Yaskawa INFORM job: DEMO_ROOF_UPPER_0625_3PAINT_23.JBI

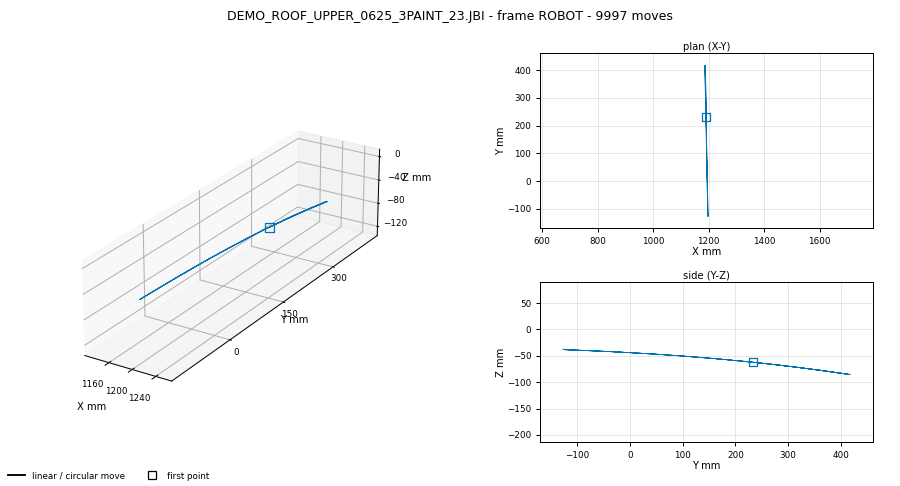
[picture p0: tool path of DEMO_ROOF_UPPER_0625_3PAINT_23.JBI in frame ROBOT, 9997 of 9997 moves have a stored position in this frame; points joined in program order, loops and branches not executed]
/JOB
//NAME DEMO_ROOF_UPPER_0625_3PAINT23
//POS
///NPOS 9997,0,0,0,0,0
///TOOL 0
///USER 0
///POSTYPE ROBOT
///RECTAN
///RCONF 1,0,0,0,0,0,0,0,0,0,0,0,0,0,0,0,0,0,0,0,0,0,0,0
C00000=1191.558,232.697,-61.990,-177.381,6.861,148.504
C00001=1191.554,232.946,-62.016,-177.379,6.863,148.503
C00002=1191.549,233.194,-62.041,-177.376,6.866,148.503
C00003=1191.545,233.443,-62.067,-177.373,6.868,148.503
C00004=1191.540,233.692,-62.093,-177.371,6.870,148.503
C00005=1191.536,233.941,-62.119,-177.368,6.873,148.503
C00006=1191.531,234.189,-62.145,-177.365,6.874,148.502
C00007=1191.527,234.437,-62.171,-177.363,6.877,148.502
C00008=1191.523,234.686,-62.197,-177.360,6.879,148.502
C00009=1191.519,234.935,-62.223,-177.358,6.881,148.502
C00010=1191.513,235.183,-62.249,-177.355,6.883,148.501
C00011=1191.509,235.432,-62.274,-177.352,6.886,148.501
C00012=1191.505,235.681,-62.300,-177.350,6.888,148.501
C00013=1191.500,235.929,-62.326,-177.348,6.890,148.501
C00014=1191.495,236.177,-62.353,-177.344,6.893,148.501
C00015=1191.490,236.449,-62.381,-177.342,6.895,148.500
C00016=1191.486,236.721,-62.409,-177.339,6.898,148.500
C00017=1191.481,236.992,-62.437,-177.336,6.900,148.500
C00018=1191.476,237.264,-62.465,-177.333,6.902,148.500
C00019=1191.471,237.512,-62.492,-177.330,6.905,148.500
C00020=1191.467,237.761,-62.518,-177.328,6.907,148.499
C00021=1191.463,238.010,-62.544,-177.326,6.909,148.499
C00022=1191.458,238.259,-62.570,-177.322,6.912,148.499
C00023=1191.453,238.506,-62.596,-177.320,6.914,148.499
C00024=1191.449,238.755,-62.622,-177.318,6.916,148.498
C00025=1191.444,239.004,-62.648,-177.315,6.919,148.498
C00026=1191.440,239.252,-62.675,-177.312,6.921,148.498
C00027=1191.436,239.501,-62.700,-177.310,6.923,148.498
C00028=1191.431,239.750,-62.727,-177.307,6.925,148.498
C00029=1191.427,239.998,-62.753,-177.305,6.928,148.498
C00030=1191.422,240.247,-62.779,-177.302,6.930,148.497
C00031=1191.418,240.495,-62.806,-177.299,6.932,148.497
C00032=1191.414,240.744,-62.831,-177.297,6.934,148.497
C00033=1191.409,240.993,-62.857,-177.294,6.937,148.497
C00034=1191.405,241.241,-62.884,-177.291,6.939,148.496
C00035=1191.400,241.490,-62.910,-177.289,6.941,148.496
C00036=1191.396,241.738,-62.937,-177.286,6.944,148.496
C00037=1191.392,241.987,-62.963,-177.284,6.946,148.496
C00038=1191.386,242.235,-62.989,-177.281,6.948,148.496
C00039=1191.382,242.484,-63.015,-177.279,6.951,148.496
C00040=1191.378,242.732,-63.042,-177.276,6.953,148.495
C00041=1191.373,242.981,-63.068,-177.273,6.956,148.495
C00042=1191.369,243.229,-63.094,-177.270,6.957,148.495
C00043=1191.364,243.478,-63.121,-177.268,6.960,148.495
C00044=1191.360,243.727,-63.147,-177.265,6.962,148.495
C00045=1191.355,243.976,-63.174,-177.263,6.964,148.494
C00046=1191.351,244.224,-63.200,-177.260,6.967,148.494
C00047=1191.347,244.473,-63.226,-177.258,6.969,148.494
C00048=1191.343,244.721,-63.253,-177.255,6.971,148.494
C00049=1191.338,244.970,-63.280,-177.252,6.974,148.494
C00050=1191.334,245.219,-63.306,-177.250,6.976,148.494
C00051=1191.329,245.467,-63.333,-177.247,6.979,148.493
C00052=1191.325,245.715,-63.359,-177.245,6.981,148.493
C00053=1191.320,245.964,-63.386,-177.242,6.983,148.493
C00054=1191.316,246.213,-63.412,-177.239,6.986,148.493
C00055=1191.312,246.461,-63.439,-177.237,6.988,148.493
C00056=1191.307,246.710,-63.465,-177.234,6.991,148.492
C00057=1191.303,246.958,-63.492,-177.231,6.992,148.492
C00058=1191.298,247.207,-63.519,-177.229,6.995,148.492
C00059=1191.294,247.456,-63.545,-177.226,6.998,148.492
C00060=1191.289,247.704,-63.572,-177.224,6.999,148.492
C00061=1191.285,247.953,-63.599,-177.221,7.002,148.492
C00062=1191.281,248.201,-63.625,-177.218,7.004,148.491
C00063=1191.276,248.450,-63.652,-177.216,7.006,148.491
C00064=1191.271,248.698,-63.679,-177.213,7.009,148.491
C00065=1191.267,248.947,-63.705,-177.211,7.011,148.491
C00066=1191.262,249.195,-63.732,-177.208,7.014,148.491
C00067=1191.258,249.443,-63.759,-177.206,7.016,148.490
C00068=1191.254,249.692,-63.786,-177.203,7.019,148.490
C00069=1191.249,249.941,-63.812,-177.200,7.021,148.490
C00070=1191.245,250.189,-63.839,-177.198,7.023,148.490
C00071=1191.240,250.438,-63.866,-177.195,7.026,148.490
C00072=1191.236,250.686,-63.893,-177.193,7.028,148.490
C00073=1191.231,250.935,-63.920,-177.190,7.031,148.490
C00074=1191.227,251.183,-63.946,-177.187,7.033,148.489
C00075=1191.222,251.431,-63.973,-177.185,7.036,148.489
C00076=1191.218,251.680,-64.000,-177.182,7.038,148.489
C00077=1191.214,251.928,-64.027,-177.179,7.041,148.489
C00078=1191.210,252.177,-64.054,-177.177,7.043,148.489
C00079=1191.205,252.426,-64.081,-177.174,7.045,148.488
C00080=1191.200,252.674,-64.108,-177.172,7.048,148.488
C00081=1191.196,252.923,-64.135,-177.170,7.050,148.488
C00082=1191.192,253.171,-64.162,-177.166,7.052,148.488
C00083=1191.187,253.419,-64.189,-177.164,7.055,148.488
C00084=1191.183,253.668,-64.216,-177.162,7.058,148.488
C00085=1191.178,253.916,-64.243,-177.159,7.059,148.488
C00086=1191.174,254.164,-64.270,-177.156,7.062,148.487
C00087=1191.170,254.414,-64.297,-177.154,7.064,148.487
C00088=1191.165,254.662,-64.324,-177.151,7.067,148.487
C00089=1191.161,254.911,-64.351,-177.149,7.069,148.487
C00090=1191.156,255.159,-64.378,-177.146,7.071,148.487
C00091=1191.151,255.408,-64.405,-177.143,7.074,148.487
C00092=1191.147,255.656,-64.432,-177.141,7.076,148.487
C00093=1191.143,255.905,-64.459,-177.138,7.079,148.486
C00094=1191.139,256.153,-64.487,-177.136,7.081,148.486
C00095=1191.134,256.401,-64.514,-177.133,7.084,148.486
C00096=1191.130,256.650,-64.541,-177.130,7.086,148.486
C00097=1191.125,256.898,-64.568,-177.128,7.089,148.486
C00098=1191.120,257.147,-64.595,-177.126,7.091,148.486
C00099=1191.117,257.395,-64.623,-177.122,7.094,148.485
C00100=1191.112,257.644,-64.650,-177.120,7.096,148.485
C00101=1191.107,257.892,-64.677,-177.117,7.099,148.485
C00102=1191.103,258.141,-64.704,-177.115,7.101,148.485
C00103=1191.099,258.388,-64.732,-177.112,7.104,148.485
C00104=1191.095,258.638,-64.759,-177.110,7.106,148.485
C00105=1191.090,258.886,-64.786,-177.107,7.109,148.485
C00106=1191.086,259.135,-64.813,-177.105,7.111,148.485
C00107=1191.081,259.383,-64.841,-177.102,7.114,148.484
C00108=1191.077,259.632,-64.868,-177.099,7.116,148.484
C00109=1191.073,259.880,-64.895,-177.097,7.119,148.484
C00110=1191.068,260.128,-64.923,-177.094,7.121,148.484
C00111=1191.064,260.377,-64.950,-177.091,7.123,148.484
C00112=1191.060,260.626,-64.978,-177.089,7.126,148.484
C00113=1191.055,260.874,-65.006,-177.086,7.129,148.484
C00114=1191.051,261.122,-65.033,-177.084,7.130,148.483
C00115=1191.046,261.370,-65.060,-177.081,7.133,148.483
C00116=1191.042,261.619,-65.088,-177.079,7.136,148.483
C00117=1191.037,261.867,-65.116,-177.076,7.139,148.483
C00118=1191.032,262.116,-65.143,-177.073,7.140,148.483
C00119=1191.028,262.389,-65.173,-177.071,7.143,148.483
C00120=1191.023,262.662,-65.204,-177.068,7.146,148.483
C00121=1191.019,262.935,-65.234,-177.065,7.149,148.482
C00122=1191.013,263.208,-65.265,-177.062,7.152,148.482
C00123=1191.009,263.456,-65.292,-177.059,7.154,148.482
C00124=1191.005,263.705,-65.320,-177.057,7.157,148.482
C00125=1191.000,263.953,-65.347,-177.055,7.159,148.482
C00126=1190.996,264.201,-65.375,-177.052,7.162,148.482
C00127=1190.992,264.450,-65.402,-177.049,7.164,148.482
C00128=1190.987,264.698,-65.430,-177.046,7.167,148.482
C00129=1190.983,264.946,-65.458,-177.044,7.169,148.481
C00130=1190.978,265.195,-65.486,-177.042,7.172,148.481
C00131=1190.974,265.443,-65.513,-177.038,7.175,148.481
C00132=1190.969,265.692,-65.540,-177.036,7.177,148.481
C00133=1190.966,265.940,-65.569,-177.034,7.180,148.481
C00134=1190.961,266.188,-65.596,-177.031,7.182,148.481
C00135=1190.956,266.437,-65.624,-177.028,7.185,148.481
C00136=1190.952,266.686,-65.652,-177.026,7.187,148.481
C00137=1190.948,266.934,-65.680,-177.023,7.190,148.481
C00138=1190.944,267.183,-65.707,-177.021,7.192,148.480
C00139=1190.939,267.431,-65.736,-177.018,7.195,148.480
C00140=1190.934,267.679,-65.764,-177.015,7.198,148.480
C00141=1190.930,267.927,-65.792,-177.013,7.200,148.480
C00142=1190.926,268.176,-65.819,-177.010,7.203,148.480
C00143=1190.921,268.425,-65.848,-177.008,7.205,148.480
C00144=1190.917,268.673,-65.875,-177.005,7.208,148.480
C00145=1190.913,268.920,-65.903,-177.003,7.210,148.480
C00146=1190.909,269.170,-65.930,-177.000,7.213,148.480
C00147=1190.903,269.418,-65.959,-176.998,7.215,148.479
C00148=1190.900,269.666,-65.987,-176.995,7.218,148.479
C00149=1190.895,269.914,-66.015,-176.992,7.221,148.479
C00150=1190.891,270.163,-66.044,-176.990,7.223,148.479
C00151=1190.887,270.411,-66.071,-176.987,7.226,148.479
C00152=1190.882,270.660,-66.099,-176.985,7.228,148.479
C00153=1190.877,270.908,-66.127,-176.982,7.231,148.479
C00154=1190.874,271.157,-66.155,-176.980,7.233,148.479
C00155=1190.869,271.405,-66.183,-176.977,7.236,148.479
C00156=1190.864,271.653,-66.211,-176.974,7.239,148.479
C00157=1190.860,271.902,-66.240,-176.972,7.241,148.478
C00158=1190.855,272.150,-66.268,-176.969,7.244,148.478
C00159=1190.852,272.398,-66.296,-176.967,7.246,148.478
C00160=1190.847,272.646,-66.324,-176.964,7.249,148.478
C00161=1190.843,272.895,-66.353,-176.961,7.252,148.478
C00162=1190.838,273.143,-66.380,-176.959,7.254,148.478
C00163=1190.834,273.392,-66.409,-176.956,7.257,148.478
C00164=1190.830,273.640,-66.437,-176.954,7.259,148.478
C00165=1190.825,273.889,-66.466,-176.951,7.262,148.478
C00166=1190.821,274.137,-66.494,-176.948,7.265,148.478
C00167=1190.817,274.385,-66.522,-176.946,7.267,148.477
C00168=1190.813,274.634,-66.550,-176.943,7.270,148.477
C00169=1190.808,274.882,-66.578,-176.941,7.272,148.477
C00170=1190.804,275.131,-66.607,-176.938,7.275,148.477
C00171=1190.799,275.379,-66.635,-176.936,7.278,148.477
C00172=1190.795,275.627,-66.664,-176.933,7.280,148.477
C00173=1190.791,275.875,-66.692,-176.931,7.283,148.477
C00174=1190.786,276.124,-66.721,-176.928,7.285,148.477
C00175=1190.783,276.372,-66.749,-176.925,7.288,148.477
C00176=1190.777,276.621,-66.777,-176.923,7.291,148.477
C00177=1190.773,276.869,-66.806,-176.920,7.293,148.477
C00178=1190.769,277.117,-66.834,-176.918,7.296,148.476
C00179=1190.764,277.366,-66.863,-176.915,7.299,148.476
C00180=1190.760,277.613,-66.891,-176.913,7.301,148.476
C00181=1190.756,277.862,-66.920,-176.910,7.304,148.476
C00182=1190.752,278.111,-66.948,-176.908,7.306,148.476
C00183=1190.747,278.358,-66.977,-176.905,7.309,148.476
C00184=1190.743,278.607,-67.005,-176.902,7.312,148.476
C00185=1190.739,278.856,-67.034,-176.900,7.314,148.476
C00186=1190.734,279.103,-67.063,-176.897,7.317,148.476
C00187=1190.730,279.352,-67.091,-176.895,7.320,148.476
C00188=1190.725,279.600,-67.119,-176.892,7.322,148.476
C00189=1190.721,279.849,-67.148,-176.889,7.325,148.475
C00190=1190.717,280.097,-67.177,-176.887,7.327,148.475
C00191=1190.712,280.345,-67.205,-176.884,7.330,148.475
C00192=1190.708,280.594,-67.235,-176.882,7.333,148.475
C00193=1190.704,280.842,-67.263,-176.879,7.335,148.475
C00194=1190.699,281.090,-67.291,-176.877,7.338,148.475
C00195=1190.695,281.339,-67.321,-176.874,7.341,148.475
C00196=1190.691,281.587,-67.349,-176.872,7.344,148.475
C00197=1190.686,281.835,-67.378,-176.869,7.347,148.475
C00198=1190.682,282.084,-67.407,-176.866,7.349,148.475
C00199=1190.678,282.332,-67.435,-176.864,7.351,148.475
C00200=1190.673,282.580,-67.464,-176.861,7.354,148.475
C00201=1190.669,282.829,-67.493,-176.858,7.357,148.475
C00202=1190.665,283.077,-67.522,-176.856,7.360,148.475
C00203=1190.661,283.325,-67.550,-176.854,7.363,148.475
C00204=1190.656,283.573,-67.579,-176.851,7.366,148.475
C00205=1190.652,283.822,-67.608,-176.849,7.368,148.474
C00206=1190.648,284.070,-67.637,-176.846,7.371,148.474
C00207=1190.643,284.318,-67.667,-176.843,7.374,148.474
C00208=1190.639,284.566,-67.695,-176.841,7.376,148.474
C00209=1190.635,284.815,-67.724,-176.838,7.379,148.474
C00210=1190.630,285.064,-67.753,-176.835,7.382,148.474
C00211=1190.626,285.311,-67.782,-176.833,7.384,148.474
C00212=1190.621,285.559,-67.811,-176.830,7.387,148.474
C00213=1190.617,285.808,-67.840,-176.828,7.390,148.474
C00214=1190.613,286.056,-67.869,-176.825,7.392,148.474
C00215=1190.608,286.304,-67.897,-176.823,7.395,148.474
C00216=1190.604,286.553,-67.927,-176.820,7.398,148.474
C00217=1190.600,286.801,-67.956,-176.818,7.400,148.474
C00218=1190.596,287.049,-67.986,-176.815,7.403,148.474
C00219=1190.591,287.298,-68.014,-176.812,7.406,148.474
C00220=1190.587,287.546,-68.044,-176.810,7.408,148.474
C00221=1190.582,287.794,-68.073,-176.808,7.411,148.474
C00222=1190.579,288.042,-68.101,-176.805,7.414,148.474
C00223=1190.573,288.317,-68.134,-176.802,7.417,148.474
C00224=1190.569,288.592,-68.166,-176.799,7.420,148.473
C00225=1190.564,288.866,-68.199,-176.796,7.423,148.473
C00226=1190.559,289.140,-68.231,-176.794,7.426,148.473
C00227=1190.555,289.388,-68.260,-176.791,7.429,148.473
C00228=1190.551,289.637,-68.290,-176.789,7.431,148.473
C00229=1190.546,289.885,-68.318,-176.786,7.434,148.473
C00230=1190.542,290.134,-68.348,-176.783,7.437,148.473
C00231=1190.538,290.382,-68.377,-176.781,7.439,148.473
C00232=1190.533,290.630,-68.406,-176.778,7.442,148.473
C00233=1190.529,290.878,-68.436,-176.776,7.445,148.473
C00234=1190.525,291.126,-68.465,-176.773,7.448,148.473
C00235=1190.521,291.374,-68.495,-176.771,7.451,148.473
C00236=1190.516,291.623,-68.524,-176.768,7.454,148.473
C00237=1190.512,291.871,-68.554,-176.765,7.457,148.473
C00238=1190.508,292.119,-68.583,-176.763,7.459,148.473
C00239=1190.504,292.367,-68.612,-176.761,7.462,148.473
C00240=1190.500,292.616,-68.642,-176.758,7.465,148.473
C00241=1190.495,292.863,-68.671,-176.755,7.468,148.473
C00242=1190.491,293.111,-68.700,-176.753,7.470,148.473
C00243=1190.487,293.360,-68.730,-176.750,7.473,148.473
C00244=1190.482,293.608,-68.759,-176.748,7.476,148.473
C00245=1190.477,293.857,-68.789,-176.745,7.478,148.472
C00246=1190.473,294.105,-68.819,-176.743,7.481,148.472
C00247=1190.469,294.353,-68.848,-176.740,7.484,148.472
C00248=1190.465,294.601,-68.878,-176.738,7.487,148.473
C00249=1190.461,294.850,-68.907,-176.736,7.490,148.473
C00250=1190.457,295.098,-68.937,-176.733,7.493,148.472
C00251=1190.452,295.346,-68.966,-176.730,7.496,148.472
C00252=1190.448,295.594,-68.996,-176.728,7.498,148.472
C00253=1190.443,295.843,-69.026,-176.725,7.501,148.472
C00254=1190.439,296.091,-69.056,-176.723,7.504,148.472
C00255=1190.435,296.339,-69.085,-176.720,7.507,148.472
C00256=1190.431,296.587,-69.115,-176.718,7.509,148.472
C00257=1190.427,296.836,-69.144,-176.715,7.512,148.472
C00258=1190.422,297.084,-69.174,-176.712,7.515,148.472
C00259=1190.418,297.332,-69.204,-176.710,7.518,148.472
C00260=1190.414,297.580,-69.234,-176.707,7.520,148.472
C00261=1190.410,297.828,-69.263,-176.705,7.523,148.472
C00262=1190.406,298.077,-69.293,-176.702,7.526,148.472
C00263=1190.401,298.324,-69.324,-176.699,7.529,148.472
C00264=1190.397,298.573,-69.353,-176.697,7.531,148.472
C00265=1190.393,298.821,-69.382,-176.695,7.535,148.472
C00266=1190.388,299.069,-69.413,-176.692,7.538,148.472
C00267=1190.384,299.317,-69.443,-176.690,7.541,148.472
C00268=1190.380,299.566,-69.472,-176.687,7.543,148.472
C00269=1190.376,299.813,-69.502,-176.685,7.546,148.472
C00270=1190.371,300.062,-69.532,-176.682,7.549,148.472
C00271=1190.367,300.310,-69.562,-176.679,7.552,148.472
C00272=1190.363,300.558,-69.592,-176.677,7.554,148.472
C00273=1190.358,300.806,-69.622,-176.674,7.557,148.472
C00274=1190.354,301.055,-69.651,-176.672,7.560,148.472
C00275=1190.350,301.302,-69.682,-176.669,7.563,148.472
C00276=1190.345,301.551,-69.712,-176.667,7.566,148.472
C00277=1190.341,301.798,-69.742,-176.665,7.569,148.472
C00278=1190.337,302.047,-69.771,-176.662,7.572,148.472
C00279=1190.332,302.295,-69.802,-176.659,7.575,148.472
C00280=1190.328,302.543,-69.832,-176.657,7.577,148.472
C00281=1190.324,302.792,-69.863,-176.654,7.580,148.472
C00282=1190.320,303.040,-69.892,-176.652,7.583,148.472
C00283=1190.315,303.288,-69.923,-176.649,7.586,148.472
C00284=1190.311,303.536,-69.952,-176.647,7.588,148.472
C00285=1190.307,303.784,-69.982,-176.644,7.591,148.472
C00286=1190.302,304.032,-70.013,-176.642,7.594,148.472
C00287=1190.298,304.280,-70.043,-176.639,7.597,148.472
C00288=1190.294,304.528,-70.073,-176.637,7.600,148.472
C00289=1190.289,304.776,-70.103,-176.634,7.603,148.472
C00290=1190.285,305.025,-70.134,-176.632,7.606,148.472
C00291=1190.281,305.273,-70.163,-176.629,7.609,148.472
C00292=1190.277,305.521,-70.194,-176.627,7.612,148.472
C00293=1190.273,305.769,-70.224,-176.624,7.614,148.472
C00294=1190.268,306.017,-70.254,-176.622,7.617,148.472
C00295=1190.264,306.265,-70.285,-176.619,7.620,148.472
C00296=1190.260,306.514,-70.316,-176.617,7.623,148.472
C00297=1190.256,306.762,-70.345,-176.615,7.626,148.472
C00298=1190.251,307.010,-70.376,-176.612,7.629,148.472
C00299=1190.247,307.257,-70.406,-176.609,7.632,148.472
C00300=1190.243,307.505,-70.437,-176.606,7.635,148.472
C00301=1190.238,307.754,-70.467,-176.604,7.638,148.472
C00302=1190.235,308.002,-70.498,-176.602,7.640,148.472
C00303=1190.230,308.250,-70.528,-176.599,7.643,148.472
C00304=1190.226,308.498,-70.558,-176.597,7.646,148.472
C00305=1190.221,308.746,-70.589,-176.594,7.649,148.472
C00306=1190.217,308.994,-70.619,-176.592,7.652,148.472
C00307=1190.213,309.243,-70.650,-176.590,7.655,148.472
C00308=1190.209,309.491,-70.681,-176.587,7.658,148.472
C00309=1190.205,309.738,-70.711,-176.584,7.661,148.472
C00310=1190.200,309.986,-70.741,-176.582,7.664,148.472
C00311=1190.196,310.235,-70.773,-176.579,7.667,148.472
C00312=1190.192,310.483,-70.803,-176.577,7.669,148.472
C00313=1190.187,310.731,-70.833,-176.574,7.672,148.472
C00314=1190.183,310.979,-70.864,-176.572,7.675,148.473
C00315=1190.179,311.228,-70.894,-176.569,7.678,148.473
C00316=1190.175,311.475,-70.925,-176.567,7.681,148.473
C00317=1190.170,311.723,-70.956,-176.565,7.684,148.472
C00318=1190.166,311.971,-70.986,-176.562,7.687,148.473
C00319=1190.162,312.220,-71.017,-176.560,7.690,148.473
C00320=1190.158,312.468,-71.048,-176.557,7.693,148.473
C00321=1190.153,312.716,-71.078,-176.554,7.696,148.473
C00322=1190.150,312.964,-71.109,-176.553,7.698,148.473
C00323=1190.145,313.212,-71.140,-176.550,7.701,148.473
C00324=1190.141,313.460,-71.171,-176.547,7.704,148.473
C00325=1190.137,313.709,-71.202,-176.544,7.707,148.473
C00326=1190.133,313.956,-71.232,-176.542,7.711,148.473
C00327=1190.127,314.232,-71.267,-176.539,7.714,148.473
C00328=1190.123,314.509,-71.301,-176.537,7.717,148.473
C00329=1190.119,314.786,-71.335,-176.534,7.720,148.473
C00330=1190.114,315.062,-71.370,-176.531,7.724,148.473
C00331=1190.110,315.310,-71.401,-176.529,7.726,148.473
C00332=1190.105,315.558,-71.431,-176.526,7.729,148.473
C00333=1190.101,315.806,-71.463,-176.524,7.733,148.473
C00334=1190.097,316.054,-71.494,-176.521,7.736,148.473
C00335=1190.093,316.302,-71.524,-176.519,7.739,148.473
C00336=1190.088,316.550,-71.555,-176.517,7.741,148.473
C00337=1190.084,316.799,-71.586,-176.514,7.744,148.473
C00338=1190.080,317.046,-71.618,-176.512,7.747,148.473
C00339=1190.075,317.294,-71.648,-176.509,7.750,148.473
C00340=1190.071,317.543,-71.680,-176.507,7.753,148.474
C00341=1190.067,317.791,-71.710,-176.504,7.756,148.474
C00342=1190.064,318.038,-71.742,-176.502,7.759,148.474
C00343=1190.059,318.286,-71.772,-176.500,7.762,148.474
C00344=1190.055,318.534,-71.803,-176.497,7.765,148.474
C00345=1190.051,318.782,-71.835,-176.495,7.768,148.474
C00346=1190.046,319.030,-71.866,-176.492,7.771,148.474
C00347=1190.042,319.279,-71.897,-176.490,7.773,148.474
C00348=1190.038,319.526,-71.928,-176.488,7.777,148.474
C00349=1190.034,319.775,-71.959,-176.485,7.780,148.474
C00350=1190.030,320.022,-71.991,-176.483,7.783,148.474
C00351=1190.026,320.271,-72.022,-176.480,7.786,148.474
C00352=1190.021,320.519,-72.053,-176.477,7.789,148.474
C00353=1190.017,320.766,-72.084,-176.476,7.792,148.474
C00354=1190.013,321.015,-72.115,-176.473,7.795,148.474
C00355=1190.008,321.262,-72.147,-176.471,7.798,148.475
C00356=1190.004,321.511,-72.178,-176.468,7.801,148.475
C00357=1190.000,321.758,-72.209,-176.465,7.804,148.475
C00358=1189.996,322.007,-72.241,-176.463,7.807,148.475
C00359=1189.992,322.254,-72.272,-176.461,7.809,148.475
C00360=1189.988,322.503,-72.303,-176.459,7.813,148.475
C00361=1189.983,322.750,-72.335,-176.456,7.816,148.475
C00362=1189.979,322.999,-72.366,-176.453,7.819,148.475
C00363=1189.975,323.246,-72.397,-176.451,7.822,148.475
C00364=1189.971,323.495,-72.428,-176.448,7.825,148.475
C00365=1189.967,323.742,-72.460,-176.446,7.828,148.475
C00366=1189.963,323.990,-72.492,-176.444,7.831,148.475
C00367=1189.958,324.238,-72.523,-176.442,7.834,148.476
C00368=1189.954,324.486,-72.555,-176.439,7.837,148.476
C00369=1189.950,324.735,-72.586,-176.437,7.840,148.476
C00370=1189.946,324.982,-72.618,-176.434,7.843,148.476
C00371=1189.942,325.231,-72.649,-176.432,7.847,148.476
C00372=1189.937,325.478,-72.680,-176.430,7.849,148.476
C00373=1189.934,325.727,-72.712,-176.427,7.852,148.476
C00374=1189.929,325.974,-72.744,-176.425,7.855,148.476
C00375=1189.925,326.222,-72.776,-176.422,7.858,148.476
C00376=1189.920,326.470,-72.807,-176.420,7.861,148.476
C00377=1189.917,326.718,-72.839,-176.417,7.865,148.477
C00378=1189.913,326.966,-72.870,-176.415,7.867,148.477
C00379=1189.909,327.214,-72.902,-176.413,7.870,148.477
C00380=1189.904,327.463,-72.934,-176.410,7.873,148.477
C00381=1189.900,327.710,-72.965,-176.408,7.877,148.477
C00382=1189.896,327.958,-72.997,-176.405,7.880,148.477
C00383=1189.892,328.206,-73.029,-176.403,7.883,148.477
C00384=1189.888,328.453,-73.060,-176.400,7.886,148.477
C00385=1189.883,328.702,-73.092,-176.399,7.888,148.477
C00386=1189.879,328.950,-73.123,-176.396,7.892,148.478
C00387=1189.875,329.198,-73.155,-176.394,7.895,148.478
C00388=1189.871,329.446,-73.187,-176.392,7.898,148.478
C00389=1189.866,329.693,-73.219,-176.389,7.901,148.478
C00390=1189.863,329.941,-73.251,-176.387,7.904,148.478
C00391=1189.859,330.189,-73.283,-176.384,7.907,148.478
C00392=1189.854,330.437,-73.315,-176.382,7.910,148.478
C00393=1189.850,330.685,-73.347,-176.380,7.913,148.478
C00394=1189.846,330.932,-73.378,-176.377,7.916,148.478
C00395=1189.841,331.181,-73.411,-176.375,7.920,148.479
C00396=1189.837,331.429,-73.442,-176.372,7.923,148.479
C00397=1189.833,331.677,-73.473,-176.370,7.926,148.479
C00398=1189.829,331.925,-73.506,-176.368,7.929,148.479
C00399=1189.825,332.173,-73.538,-176.366,7.931,148.479
C00400=1189.821,332.421,-73.570,-176.363,7.935,148.479
C00401=1189.816,332.668,-73.602,-176.361,7.938,148.479
C00402=1189.813,332.916,-73.634,-176.358,7.941,148.479
C00403=1189.808,333.165,-73.667,-176.356,7.944,148.480
C00404=1189.804,333.412,-73.698,-176.354,7.948,148.480
C00405=1189.800,333.660,-73.730,-176.351,7.951,148.480
C00406=1189.796,333.908,-73.762,-176.349,7.954,148.480
C00407=1189.792,334.156,-73.794,-176.347,7.957,148.480
C00408=1189.787,334.404,-73.826,-176.345,7.960,148.480
C00409=1189.783,334.652,-73.858,-176.342,7.963,148.480
C00410=1189.779,334.900,-73.891,-176.340,7.966,148.481
C00411=1189.775,335.147,-73.923,-176.337,7.969,148.481
C00412=1189.770,335.395,-73.955,-176.335,7.973,148.481
C00413=1189.767,335.644,-73.987,-176.333,7.976,148.481
C00414=1189.762,335.892,-74.019,-176.331,7.978,148.481
C00415=1189.758,336.139,-74.052,-176.329,7.981,148.481
C00416=1189.754,336.387,-74.084,-176.326,7.985,148.481
C00417=1189.750,336.635,-74.116,-176.324,7.988,148.482
C00418=1189.746,336.883,-74.148,-176.321,7.991,148.482
C00419=1189.742,337.130,-74.181,-176.319,7.994,148.482
C00420=1189.737,337.378,-74.213,-176.317,7.998,148.482
C00421=1189.734,337.626,-74.245,-176.315,8.001,148.482
C00422=1189.729,337.875,-74.277,-176.313,8.003,148.482
C00423=1189.726,338.122,-74.310,-176.310,8.007,148.482
C00424=1189.721,338.370,-74.342,-176.308,8.010,148.483
C00425=1189.717,338.617,-74.374,-176.306,8.013,148.483
C00426=1189.713,338.866,-74.407,-176.304,8.017,148.483
C00427=1189.708,339.114,-74.439,-176.301,8.020,148.483
C00428=1189.705,339.361,-74.472,-176.299,8.023,148.483
C00429=1189.701,339.610,-74.504,-176.296,8.026,148.484
C00430=1189.696,339.857,-74.536,-176.295,8.029,148.484
C00431=1189.691,340.136,-74.573,-176.292,8.033,148.484
C00432=1189.687,340.415,-74.610,-176.289,8.036,148.484
C00433=1189.682,340.693,-74.646,-176.287,8.039,148.484
C00434=1189.678,340.972,-74.683,-176.284,8.043,148.484
C00435=1189.673,341.220,-74.715,-176.282,8.047,148.485
C00436=1189.670,341.467,-74.748,-176.280,8.050,148.485
C00437=1189.665,341.716,-74.780,-176.278,8.053,148.485
C00438=1189.661,341.963,-74.813,-176.276,8.056,148.485
C00439=1189.657,342.212,-74.846,-176.273,8.059,148.486
C00440=1189.653,342.459,-74.878,-176.271,8.062,148.486
C00441=1189.648,342.707,-74.910,-176.268,8.065,148.486
C00442=1189.644,342.955,-74.944,-176.266,8.069,148.486
C00443=1189.641,343.203,-74.975,-176.264,8.072,148.486
C00444=1189.636,343.450,-75.009,-176.262,8.075,148.486
C00445=1189.632,343.698,-75.042,-176.260,8.079,148.487
C00446=1189.628,343.946,-75.074,-176.258,8.081,148.487
C00447=1189.624,344.194,-75.107,-176.256,8.085,148.487
C00448=1189.620,344.442,-75.140,-176.253,8.088,148.487
C00449=1189.615,344.689,-75.172,-176.251,8.091,148.487
C00450=1189.611,344.937,-75.205,-176.249,8.095,148.488
C00451=1189.607,345.185,-75.238,-176.247,8.098,148.488
C00452=1189.603,345.433,-75.270,-176.244,8.101,148.488
C00453=1189.599,345.680,-75.303,-176.242,8.105,148.488
C00454=1189.595,345.928,-75.336,-176.240,8.107,148.489
C00455=1189.591,346.177,-75.369,-176.238,8.110,148.489
C00456=1189.586,346.424,-75.402,-176.236,8.114,148.489
C00457=1189.583,346.672,-75.435,-176.234,8.117,148.489
C00458=1189.579,346.919,-75.468,-176.231,8.120,148.489
C00459=1189.574,347.168,-75.500,-176.229,8.124,148.490
C00460=1189.570,347.416,-75.533,-176.227,8.127,148.490
C00461=1189.566,347.663,-75.566,-176.225,8.130,148.490
C00462=1189.562,347.911,-75.600,-176.222,8.134,148.490
C00463=1189.558,348.159,-75.633,-176.221,8.136,148.490
C00464=1189.554,348.406,-75.666,-176.219,8.139,148.491
C00465=1189.550,348.654,-75.698,-176.216,8.143,148.491
C00466=1189.546,348.902,-75.731,-176.214,8.146,148.491
C00467=1189.542,349.150,-75.764,-176.212,8.150,148.492
C00468=1189.538,349.398,-75.797,-176.210,8.153,148.492
C00469=1189.533,349.645,-75.830,-176.208,8.156,148.492
C00470=1189.529,349.893,-75.864,-176.205,8.160,148.492
C00471=1189.525,350.141,-75.897,-176.203,8.163,148.492
C00472=1189.521,350.389,-75.930,-176.202,8.166,148.493
C00473=1189.517,350.636,-75.963,-176.199,8.169,148.493
C00474=1189.513,350.884,-75.996,-176.198,8.172,148.493
C00475=1189.509,351.132,-76.029,-176.195,8.176,148.493
C00476=1189.504,351.379,-76.063,-176.193,8.179,148.494
C00477=1189.500,351.627,-76.096,-176.191,8.182,148.494
C00478=1189.496,351.875,-76.129,-176.189,8.186,148.494
C00479=1189.492,352.123,-76.162,-176.187,8.189,148.495
C00480=1189.488,352.370,-76.195,-176.184,8.193,148.495
C00481=1189.484,352.618,-76.228,-176.183,8.195,148.495
C00482=1189.480,352.866,-76.261,-176.181,8.199,148.495
C00483=1189.476,353.114,-76.295,-176.179,8.202,148.496
C00484=1189.472,353.362,-76.328,-176.177,8.205,148.496
C00485=1189.468,353.610,-76.361,-176.174,8.209,148.496
C00486=1189.464,353.857,-76.394,-176.172,8.212,148.496
C00487=1189.460,354.105,-76.428,-176.170,8.216,148.497
C00488=1189.456,354.352,-76.461,-176.168,8.219,148.497
C00489=1189.452,354.600,-76.495,-176.166,8.222,148.497
C00490=1189.447,354.848,-76.528,-176.165,8.225,148.498
C00491=1189.443,355.096,-76.562,-176.162,8.229,148.498
C00492=1189.438,355.344,-76.595,-176.160,8.232,148.498
C00493=1189.435,355.591,-76.629,-176.158,8.235,148.498
C00494=1189.431,355.839,-76.662,-176.156,8.239,148.499
C00495=1189.427,356.087,-76.695,-176.154,8.242,148.499
C00496=1189.423,356.335,-76.728,-176.152,8.246,148.499
C00497=1189.419,356.582,-76.762,-176.150,8.249,148.500
C00498=1189.415,356.829,-76.795,-176.148,8.253,148.500
C00499=1189.410,357.077,-76.829,-176.146,8.255,148.500
C00500=1189.406,357.326,-76.863,-176.144,8.259,148.500
C00501=1189.403,357.573,-76.897,-176.142,8.262,148.501
C00502=1189.398,357.821,-76.930,-176.140,8.265,148.501
C00503=1189.394,358.068,-76.963,-176.138,8.269,148.501
C00504=1189.390,358.316,-76.997,-176.136,8.272,148.502
C00505=1189.386,358.564,-77.030,-176.134,8.276,148.502
C00506=1189.382,358.812,-77.064,-176.132,8.279,148.502
C00507=1189.378,359.059,-77.098,-176.130,8.283,148.503
C00508=1189.374,359.307,-77.131,-176.128,8.286,148.503
C00509=1189.370,359.554,-77.165,-176.127,8.289,148.503
C00510=1189.365,359.802,-77.199,-176.124,8.292,148.504
C00511=1189.362,360.050,-77.232,-176.122,8.296,148.504
C00512=1189.358,360.298,-77.266,-176.121,8.300,148.504
C00513=1189.353,360.546,-77.300,-176.118,8.303,148.505
C00514=1189.349,360.793,-77.334,-176.117,8.306,148.505
C00515=1189.346,361.041,-77.367,-176.115,8.309,148.505
C00516=1189.342,361.288,-77.401,-176.113,8.313,148.506
C00517=1189.337,361.536,-77.435,-176.111,8.316,148.506
C00518=1189.333,361.783,-77.469,-176.109,8.320,148.506
C00519=1189.330,362.032,-77.502,-176.107,8.323,148.507
C00520=1189.325,362.279,-77.537,-176.106,8.326,148.507
C00521=1189.321,362.527,-77.570,-176.104,8.330,148.507
C00522=1189.317,362.774,-77.604,-176.102,8.333,148.508
C00523=1189.313,363.023,-77.638,-176.100,8.337,148.508
C00524=1189.309,363.270,-77.672,-176.099,8.340,148.509
C00525=1189.305,363.517,-77.706,-176.097,8.343,148.509
C00526=1189.300,363.765,-77.739,-176.095,8.347,148.509
C00527=1189.297,364.013,-77.774,-176.093,8.350,148.510
C00528=1189.293,364.260,-77.807,-176.092,8.353,148.510
C00529=1189.288,364.508,-77.841,-176.090,8.357,148.511
C00530=1189.285,364.756,-77.875,-176.088,8.360,148.511
C00531=1189.281,365.004,-77.909,-176.086,8.364,148.511
C00532=1189.276,365.251,-77.943,-176.085,8.366,148.512
C00533=1189.273,365.499,-77.977,-176.083,8.370,148.512
C00534=1189.269,365.746,-78.012,-176.081,8.374,148.513
C00535=1189.264,366.027,-78.050,-176.079,8.377,148.513
C00536=1189.259,366.309,-78.088,-176.078,8.381,148.513
C00537=1189.255,366.590,-78.127,-176.076,8.384,148.514
C00538=1189.251,366.871,-78.166,-176.073,8.389,148.514
C00539=1189.247,367.119,-78.201,-176.072,8.392,148.515
C00540=1189.242,367.367,-78.234,-176.070,8.395,148.515
C00541=1189.238,367.614,-78.268,-176.069,8.399,148.516
C00542=1189.235,367.862,-78.302,-176.067,8.402,148.516
C00543=1189.230,368.109,-78.337,-176.066,8.405,148.516
C00544=1189.226,368.357,-78.370,-176.064,8.409,148.517
C00545=1189.222,368.605,-78.405,-176.063,8.412,148.517
C00546=1189.218,368.852,-78.439,-176.061,8.416,148.518
C00547=1189.214,369.100,-78.473,-176.060,8.419,148.518
C00548=1189.210,369.347,-78.507,-176.058,8.422,148.519
C00549=1189.206,369.595,-78.542,-176.056,8.426,148.519
C00550=1189.202,369.842,-78.576,-176.055,8.429,148.520
C00551=1189.198,370.091,-78.610,-176.053,8.432,148.520
C00552=1189.194,370.338,-78.644,-176.052,8.435,148.520
C00553=1189.190,370.586,-78.679,-176.051,8.439,148.521
C00554=1189.186,370.833,-78.712,-176.049,8.443,148.521
C00555=1189.181,371.080,-78.747,-176.048,8.445,148.522
C00556=1189.178,371.329,-78.782,-176.046,8.449,148.522
C00557=1189.174,371.576,-78.816,-176.045,8.452,148.523
C00558=1189.170,371.824,-78.850,-176.043,8.456,148.523
C00559=1189.166,372.071,-78.884,-176.042,8.459,148.524
C00560=1189.161,372.318,-78.919,-176.040,8.462,148.524
C00561=1189.158,372.566,-78.953,-176.039,8.465,148.525
C00562=1189.154,372.814,-78.988,-176.038,8.469,148.525
C00563=1189.150,373.062,-79.022,-176.036,8.472,148.525
C00564=1189.146,373.309,-79.056,-176.035,8.476,148.526
C00565=1189.142,373.557,-79.091,-176.034,8.478,148.526
C00566=1189.137,373.804,-79.126,-176.032,8.482,148.527
C00567=1189.133,374.051,-79.159,-176.031,8.485,148.528
C00568=1189.129,374.300,-79.194,-176.030,8.488,148.528
C00569=1189.125,374.547,-79.229,-176.028,8.492,148.528
C00570=1189.122,374.795,-79.263,-176.027,8.495,148.529
C00571=1189.117,375.042,-79.297,-176.026,8.498,148.529
C00572=1189.113,375.290,-79.333,-176.025,8.501,148.530
C00573=1189.110,375.537,-79.367,-176.023,8.504,148.530
C00574=1189.106,375.785,-79.402,-176.022,8.508,148.531
C00575=1189.101,376.032,-79.436,-176.021,8.511,148.531
C00576=1189.098,376.280,-79.470,-176.020,8.515,148.532
C00577=1189.093,376.528,-79.505,-176.018,8.518,148.532
C00578=1189.089,376.776,-79.540,-176.017,8.521,148.533
C00579=1189.086,377.022,-79.574,-176.016,8.524,148.533
C00580=1189.082,377.270,-79.609,-176.015,8.527,148.534
C00581=1189.077,377.518,-79.644,-176.014,8.531,148.535
C00582=1189.073,377.766,-79.678,-176.013,8.533,148.535
C00583=1189.069,378.013,-79.712,-176.011,8.537,148.536
C00584=1189.066,378.260,-79.748,-176.010,8.540,148.536
C00585=1189.061,378.508,-79.782,-176.009,8.543,148.537
C00586=1189.057,378.756,-79.817,-176.008,8.547,148.537
C00587=1189.053,379.003,-79.851,-176.007,8.550,148.538
C00588=1189.050,379.251,-79.886,-176.006,8.553,148.538
C00589=1189.045,379.498,-79.921,-176.005,8.556,148.539
C00590=1189.041,379.746,-79.956,-176.004,8.559,148.539
C00591=1189.037,379.993,-79.990,-176.003,8.563,148.540
C00592=1189.034,380.241,-80.025,-176.002,8.566,148.540
C00593=1189.029,380.488,-80.060,-176.001,8.569,148.541
C00594=1189.025,380.736,-80.095,-176.000,8.572,148.541
C00595=1189.021,380.983,-80.130,-175.999,8.575,148.542
C00596=1189.017,381.231,-80.165,-175.998,8.578,148.542
C00597=1189.013,381.478,-80.198,-175.997,8.581,148.543
C00598=1189.009,381.726,-80.234,-175.997,8.584,148.544
C00599=1189.005,381.973,-80.268,-175.995,8.588,148.544
C00600=1189.001,382.221,-80.303,-175.994,8.591,148.545
C00601=1188.997,382.468,-80.338,-175.993,8.594,148.545
C00602=1188.993,382.716,-80.373,-175.992,8.597,148.546
C00603=1188.990,382.963,-80.408,-175.992,8.600,148.546
C00604=1188.985,383.211,-80.443,-175.991,8.603,148.547
C00605=1188.981,383.459,-80.478,-175.990,8.606,148.548
C00606=1188.977,383.706,-80.513,-175.989,8.609,148.548
C00607=1188.973,383.954,-80.548,-175.988,8.612,148.549
C00608=1188.969,384.201,-80.583,-175.987,8.615,148.549
C00609=1188.965,384.449,-80.618,-175.986,8.618,148.550
C00610=1188.961,384.697,-80.652,-175.986,8.621,148.550
C00611=1188.957,384.943,-80.687,-175.985,8.624,148.551
C00612=1188.953,385.192,-80.722,-175.984,8.627,148.551
C00613=1188.949,385.438,-80.757,-175.984,8.630,148.552
C00614=1188.945,385.686,-80.792,-175.983,8.633,148.553
C00615=1188.941,385.934,-80.827,-175.982,8.636,148.553
C00616=1188.937,386.181,-80.862,-175.981,8.639,148.554
C00617=1188.933,386.429,-80.897,-175.981,8.642,148.554
C00618=1188.928,386.676,-80.932,-175.980,8.645,148.555
C00619=1188.925,386.924,-80.967,-175.979,8.648,148.555
C00620=1188.921,387.172,-81.002,-175.979,8.651,148.556
C00621=1188.917,387.418,-81.037,-175.978,8.654,148.557
C00622=1188.913,387.667,-81.072,-175.978,8.657,148.557
C00623=1188.910,387.914,-81.107,-175.977,8.660,148.558
C00624=1188.905,388.161,-81.142,-175.976,8.663,148.559
C00625=1188.901,388.409,-81.177,-175.976,8.665,148.559
C00626=1188.897,388.656,-81.212,-175.975,8.668,148.560
C00627=1188.893,388.904,-81.247,-175.975,8.671,148.560
C00628=1188.890,389.151,-81.283,-175.974,8.673,148.561
C00629=1188.885,389.399,-81.317,-175.973,8.677,148.561
C00630=1188.881,389.646,-81.353,-175.973,8.680,148.562
C00631=1188.878,389.894,-81.388,-175.973,8.682,148.563
C00632=1188.873,390.141,-81.423,-175.972,8.685,148.563
C00633=1188.869,390.389,-81.458,-175.971,8.688,148.564
C00634=1188.865,390.637,-81.493,-175.971,8.691,148.564
C00635=1188.861,390.884,-81.528,-175.970,8.694,148.565
C00636=1188.858,391.131,-81.564,-175.970,8.696,148.566
C00637=1188.854,391.379,-81.599,-175.970,8.699,148.566
C00638=1188.849,391.626,-81.634,-175.969,8.702,148.567
C00639=1188.845,391.910,-81.674,-175.969,8.705,148.568
C00640=1188.840,392.193,-81.715,-175.968,8.708,148.568
C00641=1188.836,392.477,-81.756,-175.968,8.712,148.569
C00642=1188.831,392.761,-81.796,-175.967,8.715,148.570
C00643=1188.827,393.008,-81.831,-175.967,8.717,148.570
C00644=1188.823,393.256,-81.866,-175.967,8.720,148.571
C00645=1188.819,393.503,-81.901,-175.966,8.723,148.571
C00646=1188.815,393.750,-81.936,-175.966,8.725,148.572
C00647=1188.811,393.998,-81.972,-175.965,8.728,148.572
C00648=1188.807,394.246,-82.007,-175.965,8.731,148.573
C00649=1188.804,394.493,-82.042,-175.965,8.733,148.574
C00650=1188.799,394.740,-82.077,-175.964,8.736,148.574
C00651=1188.795,394.988,-82.112,-175.964,8.738,148.575
C00652=1188.792,395.236,-82.148,-175.964,8.741,148.576
C00653=1188.787,395.482,-82.183,-175.963,8.744,148.576
C00654=1188.784,395.730,-82.219,-175.963,8.746,148.577
C00655=1188.780,395.978,-82.253,-175.963,8.748,148.577
C00656=1188.776,396.225,-82.289,-175.963,8.752,148.578
C00657=1188.772,396.472,-82.324,-175.962,8.754,148.579
C00658=1188.767,396.720,-82.360,-175.962,8.756,148.579
C00659=1188.763,396.968,-82.395,-175.962,8.759,148.580
C00660=1188.759,397.215,-82.430,-175.961,8.762,148.580
C00661=1188.756,397.463,-82.466,-175.961,8.764,148.581
C00662=1188.752,397.710,-82.501,-175.961,8.767,148.581
C00663=1188.748,397.957,-82.537,-175.961,8.769,148.582
C00664=1188.744,398.205,-82.571,-175.960,8.772,148.583
C00665=1188.740,398.452,-82.607,-175.960,8.774,148.583
C00666=1188.736,398.699,-82.642,-175.960,8.777,148.584
C00667=1188.732,398.947,-82.678,-175.960,8.779,148.584
C00668=1188.728,399.195,-82.714,-175.960,8.782,148.585
C00669=1188.724,399.443,-82.749,-175.959,8.784,148.586
C00670=1188.719,399.689,-82.784,-175.959,8.787,148.586
C00671=1188.716,399.937,-82.819,-175.959,8.790,148.587
C00672=1188.712,400.184,-82.855,-175.959,8.792,148.587
C00673=1188.708,400.431,-82.890,-175.958,8.794,148.588
C00674=1188.704,400.679,-82.926,-175.958,8.796,148.588
C00675=1188.700,400.927,-82.962,-175.958,8.799,148.589
C00676=1188.696,401.175,-82.997,-175.958,8.801,148.590
C00677=1188.692,401.422,-83.032,-175.958,8.803,148.590
C00678=1188.688,401.669,-83.067,-175.958,8.806,148.591
C00679=1188.684,401.917,-83.103,-175.958,8.808,148.591
C00680=1188.681,402.164,-83.138,-175.957,8.810,148.592
C00681=1188.676,402.411,-83.174,-175.957,8.813,148.592
C00682=1188.672,402.659,-83.210,-175.957,8.815,148.593
C00683=1188.668,402.906,-83.245,-175.957,8.818,148.594
C00684=1188.665,403.154,-83.281,-175.957,8.820,148.594
C00685=1188.660,403.401,-83.315,-175.957,8.822,148.595
C00686=1188.656,403.649,-83.351,-175.956,8.824,148.595
C00687=1188.653,403.896,-83.386,-175.957,8.827,148.596
C00688=1188.648,404.144,-83.423,-175.956,8.829,148.597
C00689=1188.644,404.391,-83.458,-175.956,8.831,148.597
C00690=1188.640,404.638,-83.493,-175.956,8.834,148.598
C00691=1188.637,404.886,-83.529,-175.956,8.836,148.598
C00692=1188.633,405.133,-83.564,-175.956,8.839,148.599
C00693=1188.628,405.380,-83.600,-175.956,8.841,148.599
C00694=1188.624,405.628,-83.636,-175.955,8.843,148.600
C00695=1188.621,405.875,-83.671,-175.955,8.845,148.600
C00696=1188.617,406.123,-83.707,-175.955,8.848,148.601
C00697=1188.613,406.370,-83.742,-175.955,8.850,148.602
C00698=1188.608,406.617,-83.778,-175.955,8.852,148.602
C00699=1188.605,406.865,-83.814,-175.955,8.854,148.603
C00700=1188.601,407.112,-83.849,-175.955,8.856,148.603
C00701=1188.597,407.360,-83.885,-175.955,8.858,148.604
C00702=1188.593,407.607,-83.920,-175.955,8.861,148.604
C00703=1188.589,407.854,-83.956,-175.954,8.863,148.605
C00704=1188.585,408.102,-83.992,-175.954,8.866,148.605
C00705=1188.581,408.349,-84.027,-175.955,8.867,148.606
C00706=1188.578,408.597,-84.063,-175.954,8.869,148.606
C00707=1188.573,408.844,-84.099,-175.954,8.872,148.607
C00708=1188.569,409.092,-84.134,-175.954,8.874,148.608
C00709=1188.565,409.339,-84.170,-175.954,8.876,148.608
C00710=1188.562,409.587,-84.205,-175.954,8.879,148.609
C00711=1188.557,409.834,-84.241,-175.954,8.880,148.609
C00712=1188.553,410.081,-84.277,-175.954,8.882,148.610
C00713=1188.549,410.329,-84.312,-175.954,8.885,148.610
C00714=1188.546,410.576,-84.348,-175.954,8.887,148.611
C00715=1188.541,410.824,-84.384,-175.954,8.889,148.611
C00716=1188.538,411.072,-84.419,-175.954,8.891,148.612
C00717=1188.533,411.318,-84.454,-175.953,8.893,148.613
C00718=1188.530,411.566,-84.490,-175.953,8.895,148.613
C00719=1188.525,411.814,-84.526,-175.954,8.897,148.614
C00720=1188.522,412.061,-84.562,-175.953,8.899,148.614
C00721=1188.518,412.309,-84.597,-175.953,8.901,148.615
C00722=1188.514,412.555,-84.632,-175.953,8.904,148.615
C00723=1188.509,412.803,-84.669,-175.953,8.905,148.616
C00724=1188.506,413.051,-84.704,-175.953,8.908,148.616
C00725=1188.502,413.298,-84.740,-175.953,8.910,148.617
C00726=1188.499,413.545,-84.776,-175.953,8.911,148.617
C00727=1188.494,413.792,-84.812,-175.953,8.914,148.618
C00728=1188.490,414.040,-84.847,-175.953,8.916,148.618
C00729=1188.486,414.287,-84.883,-175.953,8.918,148.619
C00730=1188.482,414.535,-84.919,-175.953,8.920,148.619
C00731=1188.478,414.783,-84.955,-175.953,8.922,148.620
C00732=1188.475,415.030,-84.990,-175.952,8.924,148.620
C00733=1188.470,415.277,-85.026,-175.953,8.925,148.621
C00734=1188.466,415.525,-85.061,-175.952,8.928,148.621
C00735=1188.460,415.924,-85.119,-175.952,8.931,148.622
C00736=1188.456,416.324,-85.177,-175.952,8.934,148.623
C00737=1188.455,416.723,-85.234,-175.952,8.937,148.624
C00738=1188.459,417.122,-85.291,-175.952,8.940,148.624
C00739=1188.038,417.123,-85.332,-175.955,8.950,148.628
C00740=1188.034,416.721,-85.275,-175.955,8.948,148.627
C00741=1188.035,416.319,-85.217,-175.956,8.945,148.627
C00742=1188.038,415.916,-85.159,-175.955,8.942,148.626
C00743=1188.045,415.513,-85.101,-175.955,8.938,148.625
C00744=1188.049,415.266,-85.065,-175.956,8.936,148.624
C00745=1188.053,415.019,-85.029,-175.955,8.935,148.624
C00746=1188.057,414.772,-84.993,-175.956,8.932,148.623
C00747=1188.061,414.524,-84.958,-175.956,8.930,148.623
C00748=1188.064,414.277,-84.922,-175.956,8.929,148.622
C00749=1188.069,414.029,-84.886,-175.956,8.926,148.622
C00750=1188.073,413.782,-84.851,-175.956,8.924,148.621
C00751=1188.077,413.534,-84.815,-175.956,8.923,148.621
C00752=1188.081,413.287,-84.779,-175.956,8.921,148.620
C00753=1188.085,413.039,-84.744,-175.956,8.918,148.620
C00754=1188.088,412.792,-84.708,-175.956,8.916,148.619
C00755=1188.092,412.545,-84.672,-175.956,8.914,148.619
C00756=1188.097,412.298,-84.636,-175.956,8.912,148.618
C00757=1188.100,412.050,-84.600,-175.956,8.910,148.618
C00758=1188.104,411.803,-84.565,-175.956,8.908,148.617
C00759=1188.108,411.555,-84.529,-175.956,8.906,148.617
C00760=1188.112,411.307,-84.493,-175.957,8.904,148.616
C00761=1188.116,411.061,-84.458,-175.957,8.902,148.616
C00762=1188.120,410.813,-84.422,-175.957,8.900,148.615
C00763=1188.124,410.565,-84.386,-175.956,8.897,148.614
C00764=1188.128,410.318,-84.351,-175.957,8.895,148.614
C00765=1188.132,410.070,-84.315,-175.957,8.893,148.613
C00766=1188.136,409.823,-84.280,-175.957,8.892,148.613
C00767=1188.140,409.576,-84.244,-175.957,8.889,148.612
C00768=1188.144,409.328,-84.208,-175.957,8.887,148.612
C00769=1188.148,409.081,-84.173,-175.957,8.885,148.611
C00770=1188.151,408.833,-84.137,-175.957,8.882,148.611
C00771=1188.156,408.586,-84.102,-175.957,8.881,148.610
C00772=1188.160,408.339,-84.066,-175.957,8.878,148.610
C00773=1188.164,408.091,-84.030,-175.957,8.876,148.609
C00774=1188.167,407.844,-83.995,-175.958,8.874,148.609
C00775=1188.171,407.596,-83.959,-175.958,8.872,148.608
C00776=1188.176,407.349,-83.924,-175.958,8.869,148.607
C00777=1188.180,407.101,-83.888,-175.957,8.868,148.607
C00778=1188.183,406.854,-83.852,-175.958,8.865,148.606
C00779=1188.187,406.606,-83.817,-175.958,8.863,148.606
C00780=1188.191,406.359,-83.781,-175.958,8.861,148.605
C00781=1188.196,406.112,-83.746,-175.958,8.858,148.605
C00782=1188.199,405.864,-83.710,-175.958,8.856,148.604
C00783=1188.203,405.617,-83.674,-175.958,8.854,148.604
C00784=1188.207,405.369,-83.639,-175.959,8.852,148.603
C00785=1188.212,405.122,-83.603,-175.958,8.849,148.602
C00786=1188.215,404.875,-83.568,-175.958,8.848,148.602
C00787=1188.219,404.627,-83.532,-175.958,8.845,148.601
C00788=1188.223,404.380,-83.497,-175.959,8.843,148.601
C00789=1188.227,404.133,-83.461,-175.958,8.840,148.600
C00790=1188.231,403.885,-83.426,-175.959,8.838,148.600
C00791=1188.235,403.638,-83.390,-175.959,8.836,148.599
C00792=1188.239,403.390,-83.354,-175.959,8.834,148.599
C00793=1188.242,403.143,-83.319,-175.959,8.831,148.598
C00794=1188.247,402.896,-83.283,-175.959,8.829,148.597
C00795=1188.251,402.648,-83.249,-175.960,8.827,148.597
C00796=1188.255,402.400,-83.212,-175.960,8.824,148.596
C00797=1188.259,402.152,-83.177,-175.960,8.822,148.595
C00798=1188.263,401.906,-83.142,-175.960,8.819,148.595
C00799=1188.267,401.658,-83.106,-175.960,8.817,148.594
C00800=1188.270,401.411,-83.071,-175.960,8.815,148.594
C00801=1188.275,401.164,-83.035,-175.960,8.812,148.593
C00802=1188.279,400.916,-82.999,-175.960,8.810,148.593
C00803=1188.283,400.668,-82.964,-175.961,8.807,148.592
C00804=1188.287,400.420,-82.929,-175.961,8.805,148.592
C00805=1188.291,400.174,-82.894,-175.961,8.802,148.591
C00806=1188.294,399.926,-82.858,-175.962,8.800,148.590
C00807=1188.298,399.679,-82.823,-175.962,8.798,148.590
C00808=1188.302,399.431,-82.787,-175.962,8.795,148.589
C00809=1188.307,399.184,-82.751,-175.962,8.793,148.589
C00810=1188.310,398.936,-82.716,-175.962,8.791,148.588
C00811=1188.314,398.688,-82.681,-175.963,8.787,148.587
C00812=1188.318,398.441,-82.645,-175.963,8.785,148.587
C00813=1188.322,398.194,-82.610,-175.963,8.783,148.586
C00814=1188.326,397.946,-82.575,-175.963,8.780,148.586
C00815=1188.330,397.699,-82.539,-175.963,8.778,148.585
C00816=1188.334,397.452,-82.505,-175.964,8.775,148.584
C00817=1188.338,397.204,-82.469,-175.964,8.772,148.584
C00818=1188.342,396.956,-82.433,-175.964,8.770,148.583
C00819=1188.346,396.709,-82.397,-175.964,8.768,148.583
C00820=1188.350,396.462,-82.362,-175.964,8.765,148.582
C00821=1188.354,396.214,-82.327,-175.965,8.762,148.581
C00822=1188.358,395.966,-82.292,-175.965,8.760,148.581
C00823=1188.362,395.720,-82.257,-175.965,8.757,148.580
C00824=1188.366,395.472,-82.221,-175.966,8.754,148.580
C00825=1188.370,395.224,-82.186,-175.966,8.752,148.579
C00826=1188.374,394.977,-82.151,-175.967,8.750,148.579
C00827=1188.378,394.730,-82.115,-175.967,8.746,148.578
C00828=1188.381,394.482,-82.080,-175.967,8.744,148.577
C00829=1188.386,394.235,-82.045,-175.967,8.742,148.577
C00830=1188.390,393.987,-82.009,-175.968,8.738,148.576
C00831=1188.394,393.739,-81.974,-175.968,8.736,148.575
C00832=1188.398,393.492,-81.938,-175.968,8.734,148.575
C00833=1188.402,393.244,-81.904,-175.969,8.731,148.574
C00834=1188.406,392.997,-81.868,-175.969,8.728,148.574
C00835=1188.410,392.749,-81.833,-175.970,8.725,148.573
C00836=1188.414,392.465,-81.793,-175.970,8.722,148.572
C00837=1188.419,392.183,-81.752,-175.970,8.719,148.572
C00838=1188.423,391.899,-81.713,-175.971,8.716,148.571
C00839=1188.428,391.616,-81.672,-175.971,8.713,148.570
C00840=1188.432,391.368,-81.637,-175.972,8.710,148.570
C00841=1188.435,391.120,-81.602,-175.973,8.708,148.569
C00842=1188.440,390.873,-81.566,-175.973,8.704,148.568
C00843=1188.444,390.625,-81.532,-175.973,8.702,148.568
C00844=1188.447,390.378,-81.496,-175.974,8.699,148.567
C00845=1188.452,390.131,-81.461,-175.974,8.697,148.567
C00846=1188.455,389.883,-81.426,-175.975,8.693,148.566
C00847=1188.459,389.635,-81.390,-175.976,8.690,148.566
C00848=1188.464,389.388,-81.356,-175.976,8.688,148.565
C00849=1188.467,389.140,-81.320,-175.976,8.685,148.564
C00850=1188.472,388.894,-81.285,-175.977,8.682,148.564
C00851=1188.476,388.645,-81.250,-175.977,8.679,148.563
C00852=1188.479,388.398,-81.215,-175.978,8.676,148.563
C00853=1188.484,388.150,-81.180,-175.979,8.673,148.562
C00854=1188.488,387.903,-81.145,-175.979,8.671,148.562
C00855=1188.491,387.655,-81.109,-175.980,8.667,148.561
C00856=1188.496,387.408,-81.075,-175.980,8.664,148.560
C00857=1188.499,387.161,-81.039,-175.981,8.661,148.560
C00858=1188.504,386.913,-81.005,-175.982,8.659,148.559
C00859=1188.508,386.666,-80.969,-175.982,8.656,148.558
C00860=1188.512,386.418,-80.934,-175.983,8.653,148.558
C00861=1188.516,386.171,-80.899,-175.984,8.650,148.557
C00862=1188.520,385.923,-80.864,-175.985,8.647,148.557
C00863=1188.524,385.675,-80.829,-175.985,8.644,148.556
C00864=1188.527,385.428,-80.795,-175.986,8.641,148.556
C00865=1188.531,385.181,-80.759,-175.987,8.638,148.555
C00866=1188.536,384.933,-80.725,-175.987,8.635,148.554
C00867=1188.539,384.686,-80.689,-175.988,8.632,148.554
C00868=1188.543,384.437,-80.655,-175.989,8.629,148.553
C00869=1188.547,384.191,-80.619,-175.990,8.626,148.553
C00870=1188.551,383.943,-80.585,-175.991,8.623,148.552
C00871=1188.556,383.695,-80.550,-175.991,8.620,148.551
C00872=1188.560,383.448,-80.515,-175.992,8.616,148.551
C00873=1188.563,383.201,-80.481,-175.993,8.613,148.550
C00874=1188.567,382.953,-80.445,-175.994,8.610,148.550
C00875=1188.571,382.705,-80.410,-175.995,8.607,148.549
C00876=1188.576,382.457,-80.376,-175.996,8.604,148.549
C00877=1188.579,382.210,-80.340,-175.997,8.601,148.548
C00878=1188.584,381.963,-80.306,-175.997,8.598,148.548
C00879=1188.588,381.715,-80.270,-175.998,8.595,148.547
C00880=1188.591,381.468,-80.236,-175.999,8.592,148.546
C00881=1188.595,381.220,-80.202,-176.000,8.589,148.546
C00882=1188.600,380.973,-80.166,-176.001,8.586,148.545
C00883=1188.604,380.725,-80.132,-176.002,8.583,148.545
C00884=1188.608,380.477,-80.097,-176.003,8.579,148.544
C00885=1188.611,380.230,-80.062,-176.004,8.576,148.544
C00886=1188.615,379.982,-80.027,-176.005,8.573,148.543
C00887=1188.620,379.735,-79.993,-176.006,8.570,148.543
C00888=1188.624,379.487,-79.958,-176.007,8.567,148.542
C00889=1188.628,379.240,-79.923,-176.008,8.563,148.541
C00890=1188.631,378.992,-79.889,-176.010,8.560,148.541
C00891=1188.636,378.745,-79.854,-176.010,8.557,148.540
C00892=1188.639,378.497,-79.819,-176.011,8.554,148.540
C00893=1188.644,378.250,-79.784,-176.012,8.551,148.540
C00894=1188.647,378.002,-79.750,-176.014,8.547,148.539
C00895=1188.652,377.754,-79.715,-176.015,8.544,148.538
C00896=1188.656,377.506,-79.681,-176.016,8.541,148.538
C00897=1188.660,377.260,-79.645,-176.017,8.538,148.537
C00898=1188.663,377.012,-79.611,-176.018,8.535,148.537
C00899=1188.668,376.764,-79.577,-176.019,8.532,148.536
C00900=1188.672,376.516,-79.542,-176.021,8.528,148.536
C00901=1188.676,376.269,-79.507,-176.022,8.525,148.535
C00902=1188.679,376.022,-79.472,-176.023,8.522,148.535
C00903=1188.684,375.774,-79.438,-176.024,8.518,148.534
C00904=1188.688,375.526,-79.403,-176.025,8.515,148.534
C00905=1188.692,375.279,-79.369,-176.026,8.512,148.533
C00906=1188.696,375.031,-79.334,-176.028,8.509,148.533
C00907=1188.700,374.783,-79.300,-176.029,8.506,148.532
C00908=1188.704,374.536,-79.266,-176.031,8.502,148.532
C00909=1188.708,374.288,-79.231,-176.032,8.499,148.531
C00910=1188.713,374.041,-79.197,-176.033,8.495,148.531
C00911=1188.715,373.794,-79.162,-176.034,8.492,148.530
C00912=1188.720,373.546,-79.127,-176.036,8.489,148.530
C00913=1188.724,373.298,-79.093,-176.037,8.486,148.529
C00914=1188.728,373.051,-79.059,-176.038,8.483,148.529
C00915=1188.732,372.803,-79.024,-176.040,8.479,148.528
C00916=1188.736,372.556,-78.990,-176.041,8.476,148.528
C00917=1188.740,372.308,-78.956,-176.043,8.472,148.527
C00918=1188.744,372.060,-78.921,-176.044,8.469,148.527
C00919=1188.748,371.813,-78.887,-176.046,8.466,148.527
C00920=1188.752,371.565,-78.852,-176.047,8.462,148.526
C00921=1188.756,371.318,-78.818,-176.048,8.459,148.526
C00922=1188.760,371.070,-78.784,-176.050,8.455,148.525
C00923=1188.764,370.822,-78.749,-176.051,8.453,148.525
C00924=1188.768,370.575,-78.715,-176.053,8.449,148.524
C00925=1188.772,370.326,-78.681,-176.054,8.446,148.524
C00926=1188.776,370.079,-78.647,-176.056,8.442,148.523
C00927=1188.781,369.832,-78.613,-176.057,8.440,148.523
C00928=1188.784,369.584,-78.578,-176.059,8.436,148.522
C00929=1188.789,369.337,-78.544,-176.060,8.432,148.522
C00930=1188.792,369.089,-78.510,-176.062,8.429,148.522
C00931=1188.796,368.841,-78.475,-176.064,8.426,148.521
C00932=1188.800,368.594,-78.441,-176.065,8.422,148.521
C00933=1188.805,368.346,-78.407,-176.066,8.419,148.520
C00934=1188.808,368.098,-78.373,-176.068,8.415,148.520
C00935=1188.813,367.851,-78.339,-176.070,8.412,148.519
C00936=1188.816,367.603,-78.305,-176.071,8.409,148.519
C00937=1188.821,367.356,-78.270,-176.073,8.405,148.518
C00938=1188.825,367.108,-78.237,-176.075,8.402,148.518
C00939=1188.829,366.860,-78.202,-176.076,8.399,148.518
C00940=1188.834,366.579,-78.164,-176.078,8.395,148.517
C00941=1188.838,366.298,-78.125,-176.080,8.391,148.517
C00942=1188.842,366.017,-78.086,-176.082,8.387,148.516
C00943=1188.848,365.735,-78.047,-176.084,8.384,148.516
C00944=1188.851,365.488,-78.014,-176.085,8.380,148.515
C00945=1188.855,365.240,-77.979,-176.087,8.377,148.515
C00946=1188.859,364.993,-77.945,-176.088,8.374,148.515
C00947=1188.863,364.745,-77.912,-176.091,8.370,148.514
C00948=1188.867,364.497,-77.877,-176.092,8.367,148.514
C00949=1188.871,364.250,-77.843,-176.094,8.364,148.514
C00950=1188.875,364.002,-77.810,-176.096,8.360,148.513
C00951=1188.879,363.754,-77.775,-176.097,8.357,148.513
C00952=1188.883,363.506,-77.742,-176.099,8.353,148.512
C00953=1188.887,363.259,-77.708,-176.101,8.350,148.512
C00954=1188.892,363.012,-77.674,-176.103,8.347,148.512
C00955=1188.895,362.763,-77.640,-176.104,8.343,148.511
C00956=1188.899,362.516,-77.606,-176.106,8.340,148.511
C00957=1188.904,362.268,-77.572,-176.108,8.336,148.511
C00958=1188.907,362.020,-77.538,-176.110,8.333,148.510
C00959=1188.911,361.773,-77.505,-176.111,8.330,148.510
C00960=1188.916,361.525,-77.471,-176.114,8.327,148.509
C00961=1188.920,361.277,-77.437,-176.116,8.323,148.509
C00962=1188.923,361.030,-77.403,-176.117,8.319,148.509
C00963=1188.928,360.782,-77.369,-176.120,8.316,148.508
C00964=1188.932,360.535,-77.336,-176.121,8.312,148.508
C00965=1188.936,360.287,-77.302,-176.123,8.310,148.508
C00966=1188.940,360.040,-77.269,-176.125,8.306,148.507
C00967=1188.944,359.791,-77.234,-176.127,8.303,148.507
C00968=1188.948,359.544,-77.201,-176.129,8.299,148.507
C00969=1188.952,359.296,-77.167,-176.131,8.296,148.506
C00970=1188.956,359.049,-77.134,-176.133,8.292,148.506
C00971=1188.960,358.801,-77.100,-176.135,8.289,148.506
C00972=1188.965,358.553,-77.066,-176.136,8.286,148.505
C00973=1188.968,358.305,-77.032,-176.138,8.283,148.505
C00974=1188.973,358.058,-76.999,-176.140,8.279,148.505
C00975=1188.977,357.810,-76.966,-176.142,8.276,148.504
C00976=1188.981,357.563,-76.932,-176.145,8.272,148.504
C00977=1188.985,357.314,-76.898,-176.146,8.269,148.504
C00978=1188.989,357.066,-76.865,-176.149,8.265,148.503
C00979=1188.993,356.819,-76.831,-176.151,8.262,148.503
C00980=1188.997,356.572,-76.798,-176.153,8.258,148.503
C00981=1189.001,356.324,-76.765,-176.154,8.256,148.503
C00982=1189.005,356.076,-76.732,-176.156,8.252,148.502
C00983=1189.009,355.828,-76.697,-176.158,8.249,148.502
C00984=1189.013,355.580,-76.664,-176.161,8.246,148.502
C00985=1189.017,355.332,-76.630,-176.162,8.242,148.501
C00986=1189.022,355.085,-76.597,-176.165,8.239,148.501
C00987=1189.025,354.838,-76.563,-176.167,8.235,148.501
C00988=1189.030,354.590,-76.530,-176.169,8.232,148.500
C00989=1189.034,354.342,-76.497,-176.171,8.228,148.500
C00990=1189.038,354.094,-76.464,-176.173,8.225,148.500
C00991=1189.042,353.847,-76.431,-176.174,8.222,148.500
C00992=1189.045,353.598,-76.397,-176.177,8.219,148.499
C00993=1189.050,353.351,-76.364,-176.179,8.216,148.499
C00994=1189.054,353.103,-76.330,-176.181,8.212,148.499
C00995=1189.058,352.855,-76.296,-176.183,8.209,148.498
C00996=1189.062,352.608,-76.263,-176.185,8.205,148.498
C00997=1189.067,352.360,-76.230,-176.187,8.202,148.498
C00998=1189.071,352.112,-76.197,-176.190,8.199,148.498
C00999=1189.075,351.865,-76.164,-176.191,8.195,148.497
C01000=1189.079,351.617,-76.131,-176.194,8.192,148.497
C01001=1189.083,351.369,-76.098,-176.195,8.189,148.497
C01002=1189.087,351.121,-76.064,-176.198,8.186,148.497
C01003=1189.091,350.874,-76.031,-176.200,8.183,148.497
C01004=1189.096,350.626,-75.998,-176.202,8.179,148.496
C01005=1189.100,350.378,-75.965,-176.204,8.176,148.496
C01006=1189.104,350.130,-75.932,-176.206,8.172,148.496
C01007=1189.107,349.883,-75.899,-176.208,8.169,148.495
C01008=1189.111,349.635,-75.866,-176.211,8.166,148.495
C01009=1189.115,349.387,-75.833,-176.213,8.162,148.495
C01010=1189.119,349.139,-75.799,-176.215,8.159,148.495
C01011=1189.124,348.891,-75.767,-176.217,8.157,148.495
C01012=1189.128,348.643,-75.734,-176.219,8.153,148.494
C01013=1189.132,348.395,-75.701,-176.221,8.150,148.494
C01014=1189.136,348.148,-75.667,-176.223,8.146,148.494
C01015=1189.140,347.900,-75.634,-176.225,8.143,148.494
C01016=1189.144,347.652,-75.601,-176.228,8.140,148.493
C01017=1189.149,347.405,-75.568,-176.230,8.136,148.493
C01018=1189.153,347.157,-75.537,-176.232,8.133,148.493
C01019=1189.157,346.909,-75.503,-176.234,8.130,148.493
C01020=1189.161,346.662,-75.470,-176.236,8.127,148.492
C01021=1189.165,346.414,-75.437,-176.238,8.124,148.492
C01022=1189.169,346.166,-75.405,-176.241,8.121,148.492
C01023=1189.174,345.918,-75.371,-176.243,8.117,148.492
C01024=1189.178,345.670,-75.338,-176.245,8.114,148.492
C01025=1189.181,345.423,-75.306,-176.247,8.111,148.491
C01026=1189.186,345.174,-75.273,-176.250,8.107,148.491
C01027=1189.190,344.927,-75.240,-176.252,8.104,148.491
C01028=1189.194,344.679,-75.207,-176.254,8.101,148.491
C01029=1189.198,344.430,-75.175,-176.256,8.098,148.491
C01030=1189.202,344.183,-75.142,-176.258,8.095,148.490
C01031=1189.206,343.935,-75.109,-176.260,8.091,148.490
C01032=1189.210,343.687,-75.076,-176.262,8.088,148.490
C01033=1189.215,343.440,-75.044,-176.265,8.085,148.490
C01034=1189.219,343.192,-75.012,-176.267,8.081,148.489
C01035=1189.223,342.944,-74.979,-176.269,8.078,148.489
C01036=1189.227,342.696,-74.945,-176.271,8.075,148.489
C01037=1189.231,342.448,-74.913,-176.274,8.071,148.489
C01038=1189.235,342.201,-74.880,-176.276,8.069,148.489
C01039=1189.239,341.952,-74.848,-176.278,8.066,148.489
C01040=1189.243,341.705,-74.815,-176.280,8.063,148.488
C01041=1189.248,341.457,-74.783,-176.283,8.059,148.488
C01042=1189.252,341.210,-74.750,-176.285,8.056,148.488
C01043=1189.256,340.961,-74.718,-176.287,8.053,148.488
C01044=1189.261,340.683,-74.681,-176.289,8.049,148.488
C01045=1189.265,340.404,-74.645,-176.293,8.046,148.487
C01046=1189.270,340.126,-74.608,-176.295,8.042,148.487
C01047=1189.274,339.847,-74.572,-176.297,8.039,148.487
C01048=1189.279,339.599,-74.539,-176.299,8.036,148.487
C01049=1189.283,339.350,-74.507,-176.302,8.032,148.487
C01050=1189.286,339.103,-74.474,-176.304,8.029,148.486
C01051=1189.292,338.855,-74.442,-176.307,8.026,148.486
C01052=1189.295,338.608,-74.409,-176.309,8.023,148.486
C01053=1189.299,338.359,-74.377,-176.311,8.019,148.486
C01054=1189.304,338.111,-74.345,-176.313,8.016,148.486
C01055=1189.307,337.864,-74.312,-176.315,8.013,148.486
C01056=1189.312,337.616,-74.280,-176.318,8.010,148.486
C01057=1189.316,337.368,-74.248,-176.320,8.007,148.485
C01058=1189.320,337.120,-74.215,-176.322,8.004,148.485
C01059=1189.324,336.872,-74.183,-176.324,8.000,148.485
C01060=1189.328,336.624,-74.151,-176.327,7.997,148.485
C01061=1189.333,336.377,-74.119,-176.329,7.994,148.485
C01062=1189.337,336.129,-74.086,-176.332,7.991,148.484
C01063=1189.340,335.881,-74.054,-176.333,7.988,148.484
C01064=1189.345,335.632,-74.022,-176.336,7.985,148.484
C01065=1189.349,335.385,-73.990,-176.338,7.982,148.484
C01066=1189.354,335.137,-73.958,-176.340,7.979,148.484
C01067=1189.357,334.889,-73.925,-176.343,7.976,148.484
C01068=1189.361,334.641,-73.893,-176.345,7.972,148.484
C01069=1189.366,334.394,-73.861,-176.348,7.969,148.483
C01070=1189.370,334.145,-73.829,-176.350,7.966,148.483
C01071=1189.374,333.897,-73.797,-176.352,7.963,148.483
C01072=1189.378,333.649,-73.765,-176.354,7.960,148.483
C01073=1189.383,333.402,-73.733,-176.357,7.957,148.483
C01074=1189.386,333.154,-73.701,-176.359,7.954,148.483
C01075=1189.390,332.906,-73.668,-176.361,7.950,148.483
C01076=1189.395,332.658,-73.637,-176.364,7.947,148.483
C01077=1189.399,332.410,-73.604,-176.366,7.944,148.482
C01078=1189.403,332.162,-73.572,-176.369,7.941,148.482
C01079=1189.407,331.915,-73.541,-176.371,7.939,148.482
C01080=1189.412,331.666,-73.508,-176.373,7.935,148.482
C01081=1189.415,331.418,-73.477,-176.375,7.932,148.482
C01082=1189.420,331.171,-73.445,-176.378,7.929,148.482
C01083=1189.424,330.923,-73.413,-176.380,7.926,148.482
C01084=1189.428,330.675,-73.381,-176.383,7.923,148.482
C01085=1189.432,330.427,-73.349,-176.385,7.919,148.481
C01086=1189.437,330.179,-73.317,-176.387,7.917,148.481
C01087=1189.440,329.931,-73.285,-176.390,7.914,148.481
C01088=1189.445,329.683,-73.254,-176.392,7.910,148.481
C01089=1189.449,329.435,-73.222,-176.395,7.907,148.481
C01090=1189.453,329.186,-73.190,-176.397,7.904,148.481
C01091=1189.457,328.939,-73.159,-176.399,7.901,148.481
C01092=1189.461,328.691,-73.127,-176.402,7.898,148.481
C01093=1189.466,328.443,-73.095,-176.403,7.895,148.480
C01094=1189.470,328.195,-73.063,-176.406,7.892,148.480
C01095=1189.474,327.947,-73.032,-176.408,7.889,148.480
C01096=1189.478,327.699,-73.000,-176.411,7.886,148.480
C01097=1189.483,327.451,-72.968,-176.413,7.883,148.480
C01098=1189.487,327.204,-72.936,-176.416,7.880,148.480
C01099=1189.491,326.956,-72.904,-176.418,7.876,148.480
C01100=1189.495,326.707,-72.873,-176.420,7.874,148.480
C01101=1189.499,326.460,-72.842,-176.423,7.871,148.480
C01102=1189.503,326.211,-72.809,-176.425,7.868,148.480
C01103=1189.508,325.964,-72.778,-176.428,7.864,148.479
C01104=1189.512,325.715,-72.747,-176.430,7.861,148.479
C01105=1189.516,325.468,-72.715,-176.433,7.858,148.479
C01106=1189.520,325.220,-72.683,-176.435,7.855,148.479
C01107=1189.524,324.971,-72.652,-176.437,7.853,148.479
C01108=1189.528,324.724,-72.621,-176.440,7.850,148.479
C01109=1189.532,324.476,-72.588,-176.442,7.846,148.479
C01110=1189.537,324.228,-72.558,-176.445,7.843,148.479
C01111=1189.541,323.980,-72.526,-176.447,7.840,148.479
C01112=1189.545,323.732,-72.494,-176.450,7.837,148.479
C01113=1189.549,323.484,-72.463,-176.452,7.834,148.478
C01114=1189.553,323.236,-72.432,-176.454,7.831,148.479
C01115=1189.557,322.988,-72.401,-176.456,7.828,148.478
C01116=1189.562,322.740,-72.369,-176.459,7.825,148.478
C01117=1189.566,322.492,-72.338,-176.462,7.822,148.478
C01118=1189.570,322.244,-72.306,-176.464,7.819,148.478
C01119=1189.574,321.996,-72.275,-176.467,7.816,148.478
C01120=1189.578,321.748,-72.244,-176.468,7.813,148.478
C01121=1189.582,321.500,-72.213,-176.471,7.810,148.478
C01122=1189.587,321.252,-72.181,-176.474,7.807,148.478
C01123=1189.591,321.004,-72.150,-176.476,7.804,148.478
C01124=1189.595,320.756,-72.119,-176.479,7.801,148.478
C01125=1189.599,320.508,-72.087,-176.481,7.798,148.478
C01126=1189.603,320.260,-72.056,-176.483,7.795,148.478
C01127=1189.607,320.012,-72.025,-176.485,7.792,148.477
C01128=1189.612,319.764,-71.993,-176.488,7.789,148.477
C01129=1189.616,319.516,-71.962,-176.491,7.786,148.477
C01130=1189.620,319.268,-71.931,-176.493,7.783,148.477
C01131=1189.625,319.020,-71.900,-176.496,7.780,148.477
C01132=1189.629,318.772,-71.869,-176.498,7.778,148.477
C01133=1189.633,318.524,-71.838,-176.500,7.774,148.477
C01134=1189.637,318.276,-71.806,-176.503,7.771,148.477
C01135=1189.642,318.028,-71.775,-176.505,7.768,148.477
C01136=1189.646,317.780,-71.745,-176.508,7.765,148.477
C01137=1189.650,317.532,-71.713,-176.510,7.762,148.477
C01138=1189.654,317.284,-71.683,-176.512,7.759,148.477
C01139=1189.658,317.035,-71.652,-176.515,7.756,148.477
C01140=1189.662,316.788,-71.621,-176.517,7.753,148.477
C01141=1189.667,316.540,-71.589,-176.520,7.750,148.477
C01142=1189.671,316.292,-71.558,-176.522,7.747,148.477
C01143=1189.675,316.044,-71.527,-176.525,7.744,148.477
C01144=1189.679,315.795,-71.496,-176.527,7.742,148.476
C01145=1189.683,315.547,-71.466,-176.529,7.739,148.476
C01146=1189.688,315.300,-71.435,-176.532,7.736,148.476
C01147=1189.692,315.051,-71.404,-176.535,7.733,148.476
C01148=1189.697,314.775,-71.370,-176.537,7.729,148.476
C01149=1189.702,314.498,-71.335,-176.540,7.726,148.476
C01150=1189.706,314.222,-71.300,-176.543,7.722,148.476
C01151=1189.711,313.945,-71.267,-176.546,7.719,148.476
C01152=1189.715,313.697,-71.236,-176.548,7.716,148.476
C01153=1189.719,313.448,-71.205,-176.550,7.714,148.476
C01154=1189.723,313.201,-71.174,-176.553,7.711,148.476
C01155=1189.728,312.954,-71.143,-176.556,7.708,148.476
C01156=1189.732,312.705,-71.112,-176.558,7.705,148.476
C01157=1189.736,312.457,-71.081,-176.561,7.702,148.476
C01158=1189.740,312.209,-71.051,-176.563,7.699,148.476
C01159=1189.745,311.961,-71.020,-176.565,7.696,148.476
C01160=1189.749,311.713,-70.989,-176.568,7.693,148.476
C01161=1189.753,311.465,-70.959,-176.570,7.690,148.476
C01162=1189.757,311.217,-70.928,-176.573,7.687,148.476
C01163=1189.762,310.969,-70.897,-176.575,7.684,148.476
C01164=1189.765,310.720,-70.868,-176.577,7.681,148.476
C01165=1189.770,310.472,-70.837,-176.580,7.678,148.476
C01166=1189.775,310.224,-70.806,-176.583,7.675,148.476
C01167=1189.778,309.977,-70.776,-176.585,7.672,148.475
C01168=1189.783,309.728,-70.745,-176.588,7.669,148.475
C01169=1189.787,309.480,-70.714,-176.590,7.667,148.476
C01170=1189.791,309.232,-70.684,-176.593,7.664,148.476
C01171=1189.796,308.984,-70.653,-176.595,7.661,148.476
C01172=1189.800,308.735,-70.623,-176.598,7.658,148.475
C01173=1189.804,308.487,-70.592,-176.600,7.655,148.475
C01174=1189.808,308.239,-70.562,-176.602,7.652,148.475
C01175=1189.812,307.992,-70.531,-176.605,7.649,148.475
C01176=1189.817,307.744,-70.501,-176.607,7.646,148.475
C01177=1189.820,307.495,-70.471,-176.610,7.643,148.475
C01178=1189.825,307.247,-70.440,-176.612,7.641,148.475
C01179=1189.830,306.999,-70.409,-176.615,7.638,148.475
C01180=1189.834,306.751,-70.379,-176.618,7.635,148.475
C01181=1189.839,306.503,-70.349,-176.620,7.632,148.475
C01182=1189.842,306.254,-70.319,-176.623,7.629,148.475
C01183=1189.846,306.006,-70.288,-176.625,7.626,148.475
C01184=1189.851,305.758,-70.258,-176.628,7.623,148.475
C01185=1189.855,305.510,-70.228,-176.630,7.620,148.475
C01186=1189.859,305.263,-70.197,-176.633,7.617,148.475
C01187=1189.864,305.014,-70.167,-176.635,7.614,148.475
C01188=1189.868,304.766,-70.137,-176.637,7.612,148.475
C01189=1189.872,304.518,-70.106,-176.640,7.609,148.475
C01190=1189.876,304.269,-70.077,-176.643,7.606,148.475
C01191=1189.881,304.021,-70.046,-176.645,7.603,148.475
C01192=1189.885,303.773,-70.016,-176.648,7.601,148.475
C01193=1189.889,303.525,-69.986,-176.650,7.598,148.475
C01194=1189.894,303.277,-69.956,-176.653,7.594,148.475
C01195=1189.898,303.029,-69.926,-176.655,7.591,148.475
C01196=1189.902,302.781,-69.896,-176.657,7.589,148.475
C01197=1189.906,302.533,-69.866,-176.660,7.586,148.475
C01198=1189.911,302.284,-69.835,-176.663,7.583,148.475
C01199=1189.915,302.036,-69.805,-176.666,7.580,148.475
C01200=1189.919,301.788,-69.776,-176.668,7.577,148.475
C01201=1189.923,301.540,-69.745,-176.670,7.575,148.475
C01202=1189.927,301.292,-69.716,-176.673,7.572,148.475
C01203=1189.932,301.044,-69.685,-176.675,7.569,148.475
C01204=1189.936,300.795,-69.655,-176.678,7.566,148.475
C01205=1189.940,300.548,-69.625,-176.680,7.564,148.475
C01206=1189.945,300.299,-69.595,-176.683,7.560,148.475
C01207=1189.949,300.051,-69.566,-176.686,7.557,148.475
C01208=1189.953,299.803,-69.536,-176.688,7.554,148.475
C01209=1189.957,299.555,-69.506,-176.690,7.552,148.475
C01210=1189.962,299.306,-69.476,-176.693,7.549,148.475
C01211=1189.966,299.059,-69.446,-176.695,7.546,148.475
C01212=1189.970,298.811,-69.416,-176.698,7.543,148.475
C01213=1189.975,298.562,-69.386,-176.700,7.541,148.475
C01214=1189.979,298.314,-69.356,-176.703,7.538,148.475
C01215=1189.983,298.066,-69.327,-176.706,7.535,148.475
C01216=1189.987,297.818,-69.297,-176.708,7.532,148.475
C01217=1189.992,297.569,-69.267,-176.711,7.530,148.475
C01218=1189.996,297.322,-69.237,-176.713,7.527,148.475
C01219=1190.000,297.073,-69.208,-176.716,7.524,148.475
C01220=1190.005,296.825,-69.178,-176.719,7.521,148.475
C01221=1190.009,296.577,-69.149,-176.721,7.518,148.476
C01222=1190.014,296.328,-69.119,-176.724,7.515,148.476
C01223=1190.018,296.081,-69.088,-176.726,7.512,148.475
C01224=1190.022,295.832,-69.059,-176.729,7.509,148.475
C01225=1190.026,295.584,-69.030,-176.731,7.507,148.475
C01226=1190.030,295.336,-69.000,-176.733,7.504,148.475
C01227=1190.034,295.087,-68.971,-176.736,7.501,148.476
C01228=1190.039,294.839,-68.941,-176.738,7.499,148.476
C01229=1190.043,294.591,-68.911,-176.741,7.496,148.476
C01230=1190.047,294.343,-68.881,-176.744,7.493,148.476
C01231=1190.051,294.095,-68.852,-176.746,7.490,148.476
C01232=1190.056,293.846,-68.822,-176.749,7.488,148.476
C01233=1190.060,293.598,-68.793,-176.751,7.485,148.476
C01234=1190.064,293.350,-68.763,-176.754,7.482,148.476
C01235=1190.068,293.102,-68.734,-176.757,7.479,148.476
C01236=1190.072,292.853,-68.704,-176.759,7.476,148.476
C01237=1190.077,292.605,-68.674,-176.762,7.473,148.476
C01238=1190.082,292.357,-68.645,-176.764,7.470,148.476
C01239=1190.086,292.109,-68.616,-176.766,7.468,148.476
C01240=1190.090,291.861,-68.586,-176.769,7.465,148.476
C01241=1190.095,291.612,-68.557,-176.772,7.462,148.476
C01242=1190.099,291.364,-68.527,-176.775,7.459,148.476
C01243=1190.103,291.116,-68.498,-176.777,7.457,148.476
C01244=1190.107,290.867,-68.469,-176.779,7.454,148.476
C01245=1190.112,290.619,-68.440,-176.782,7.451,148.476
C01246=1190.116,290.371,-68.411,-176.784,7.449,148.476
C01247=1190.121,290.123,-68.381,-176.787,7.446,148.476
C01248=1190.125,289.875,-68.352,-176.790,7.443,148.476
C01249=1190.129,289.626,-68.322,-176.792,7.441,148.476
C01250=1190.133,289.378,-68.293,-176.795,7.438,148.476
C01251=1190.138,289.129,-68.264,-176.797,7.435,148.476
C01252=1190.142,288.855,-68.232,-176.800,7.432,148.476
C01253=1190.147,288.581,-68.200,-176.803,7.429,148.477
C01254=1190.152,288.306,-68.167,-176.805,7.426,148.477
C01255=1190.156,288.032,-68.135,-176.808,7.423,148.477
C01256=1190.161,287.784,-68.106,-176.811,7.420,148.477
C01257=1190.165,287.535,-68.077,-176.814,7.417,148.477
C01258=1190.169,287.287,-68.047,-176.816,7.415,148.477
C01259=1190.174,287.039,-68.018,-176.819,7.412,148.477
C01260=1190.178,286.791,-67.989,-176.822,7.409,148.477
C01261=1190.183,286.542,-67.960,-176.824,7.407,148.477
C01262=1190.187,286.294,-67.931,-176.826,7.404,148.477
C01263=1190.191,286.046,-67.902,-176.829,7.401,148.477
C01264=1190.195,285.797,-67.873,-176.831,7.398,148.477
C01265=1190.200,285.549,-67.844,-176.834,7.395,148.477
C01266=1190.204,285.301,-67.815,-176.837,7.392,148.477
C01267=1190.209,285.053,-67.786,-176.839,7.390,148.477
C01268=1190.213,284.804,-67.757,-176.842,7.387,148.477
C01269=1190.217,284.556,-67.729,-176.844,7.384,148.477
C01270=1190.221,284.308,-67.699,-176.846,7.382,148.477
C01271=1190.226,284.059,-67.671,-176.849,7.379,148.477
C01272=1190.230,283.811,-67.641,-176.852,7.376,148.478
C01273=1190.234,283.563,-67.612,-176.854,7.374,148.478
C01274=1190.238,283.314,-67.584,-176.857,7.371,148.478
C01275=1190.243,283.067,-67.555,-176.860,7.368,148.478
C01276=1190.247,282.818,-67.526,-176.862,7.366,148.478
C01277=1190.252,282.570,-67.496,-176.865,7.363,148.478
C01278=1190.256,282.322,-67.469,-176.868,7.360,148.478
C01279=1190.260,282.073,-67.439,-176.870,7.358,148.478
C01280=1190.265,281.825,-67.410,-176.872,7.355,148.478
C01281=1190.269,281.577,-67.383,-176.875,7.352,148.478
C01282=1190.273,281.328,-67.353,-176.877,7.350,148.478
C01283=1190.278,281.079,-67.325,-176.880,7.347,148.478
C01284=1190.282,280.832,-67.295,-176.883,7.344,148.478
C01285=1190.286,280.583,-67.267,-176.885,7.342,148.478
C01286=1190.291,280.334,-67.239,-176.888,7.339,148.479
C01287=1190.295,280.087,-67.209,-176.891,7.336,148.479
C01288=1190.299,279.838,-67.181,-176.893,7.334,148.479
C01289=1190.304,279.589,-67.153,-176.896,7.331,148.479
C01290=1190.308,279.342,-67.124,-176.898,7.328,148.479
C01291=1190.312,279.093,-67.095,-176.900,7.326,148.479
C01292=1190.317,278.844,-67.067,-176.903,7.323,148.479
C01293=1190.321,278.597,-67.038,-176.905,7.320,148.479
C01294=1190.325,278.348,-67.009,-176.909,7.318,148.479
C01295=1190.330,278.099,-66.981,-176.911,7.315,148.479
C01296=1190.334,277.851,-66.953,-176.913,7.313,148.479
C01297=1190.338,277.603,-66.923,-176.916,7.310,148.479
C01298=1190.343,277.355,-66.896,-176.919,7.307,148.479
C01299=1190.347,277.106,-66.867,-176.921,7.304,148.480
C01300=1190.351,276.858,-66.839,-176.924,7.301,148.480
C01301=1190.356,276.610,-66.810,-176.926,7.299,148.480
C01302=1190.359,276.362,-66.782,-176.929,7.297,148.480
C01303=1190.364,276.114,-66.753,-176.932,7.294,148.480
C01304=1190.368,275.865,-66.725,-176.934,7.291,148.480
C01305=1190.373,275.617,-66.697,-176.937,7.288,148.480
C01306=1190.377,275.368,-66.669,-176.939,7.285,148.480
C01307=1190.382,275.119,-66.640,-176.942,7.283,148.480
C01308=1190.386,274.871,-66.612,-176.945,7.281,148.480
C01309=1190.390,274.623,-66.583,-176.947,7.278,148.480
C01310=1190.394,274.375,-66.555,-176.950,7.275,148.481
C01311=1190.399,274.126,-66.526,-176.952,7.272,148.481
C01312=1190.403,273.879,-66.498,-176.954,7.270,148.481
C01313=1190.408,273.630,-66.470,-176.957,7.267,148.481
C01314=1190.412,273.382,-66.442,-176.960,7.265,148.481
C01315=1190.417,273.133,-66.413,-176.962,7.262,148.481
C01316=1190.421,272.885,-66.385,-176.965,7.259,148.481
C01317=1190.425,272.636,-66.356,-176.967,7.257,148.481
C01318=1190.430,272.388,-66.329,-176.970,7.254,148.481
C01319=1190.434,272.140,-66.301,-176.972,7.252,148.481
C01320=1190.439,271.891,-66.272,-176.975,7.249,148.482
C01321=1190.442,271.643,-66.244,-176.978,7.246,148.482
C01322=1190.447,271.395,-66.216,-176.980,7.244,148.482
C01323=1190.452,271.146,-66.188,-176.983,7.241,148.482
C01324=1190.456,270.898,-66.160,-176.985,7.239,148.482
C01325=1190.460,270.649,-66.132,-176.988,7.236,148.482
C01326=1190.465,270.401,-66.104,-176.991,7.234,148.482
C01327=1190.468,270.152,-66.076,-176.993,7.231,148.482
C01328=1190.474,269.904,-66.047,-176.996,7.228,148.482
C01329=1190.478,269.656,-66.020,-176.998,7.226,148.482
C01330=1190.482,269.408,-65.992,-177.001,7.223,148.483
C01331=1190.487,269.159,-65.964,-177.003,7.221,148.483
C01332=1190.491,268.910,-65.936,-177.006,7.218,148.483
C01333=1190.495,268.662,-65.908,-177.009,7.215,148.483
C01334=1190.499,268.414,-65.880,-177.012,7.213,148.483
C01335=1190.504,268.165,-65.852,-177.014,7.210,148.483
C01336=1190.509,267.917,-65.824,-177.016,7.208,148.483
C01337=1190.512,267.669,-65.796,-177.019,7.205,148.483
C01338=1190.517,267.421,-65.768,-177.021,7.203,148.483
C01339=1190.522,267.171,-65.740,-177.024,7.200,148.484
C01340=1190.526,266.923,-65.713,-177.027,7.198,148.484
C01341=1190.530,266.675,-65.685,-177.029,7.195,148.484
C01342=1190.534,266.426,-65.657,-177.032,7.192,148.484
C01343=1190.539,266.178,-65.629,-177.035,7.190,148.484
C01344=1190.543,265.929,-65.601,-177.037,7.187,148.484
C01345=1190.548,265.681,-65.574,-177.040,7.185,148.484
C01346=1190.552,265.433,-65.546,-177.042,7.182,148.484
C01347=1190.556,265.185,-65.518,-177.045,7.180,148.484
C01348=1190.561,264.936,-65.490,-177.048,7.177,148.485
C01349=1190.566,264.688,-65.463,-177.050,7.175,148.485
C01350=1190.570,264.439,-65.435,-177.053,7.172,148.485
C01351=1190.574,264.191,-65.407,-177.055,7.170,148.485
C01352=1190.578,263.943,-65.380,-177.058,7.167,148.485
C01353=1190.582,263.694,-65.352,-177.061,7.164,148.485
C01354=1190.587,263.446,-65.324,-177.063,7.162,148.485
C01355=1190.592,263.197,-65.297,-177.066,7.160,148.485
C01356=1190.596,262.924,-65.267,-177.068,7.157,148.485
C01357=1190.601,262.651,-65.236,-177.071,7.155,148.486
C01358=1190.606,262.378,-65.206,-177.074,7.152,148.486
C01359=1190.611,262.106,-65.176,-177.077,7.149,148.486
C01360=1190.616,261.857,-65.148,-177.080,7.146,148.486
C01361=1190.620,261.608,-65.120,-177.082,7.144,148.486
C01362=1190.624,261.360,-65.093,-177.085,7.141,148.486
C01363=1190.629,261.112,-65.065,-177.087,7.139,148.487
C01364=1190.633,260.863,-65.038,-177.090,7.136,148.487
C01365=1190.637,260.614,-65.011,-177.092,7.134,148.487
C01366=1190.642,260.366,-64.983,-177.095,7.131,148.487
C01367=1190.646,260.118,-64.956,-177.098,7.129,148.487
C01368=1190.651,259.870,-64.928,-177.100,7.126,148.487
C01369=1190.655,259.621,-64.901,-177.103,7.124,148.487
C01370=1190.660,259.372,-64.874,-177.106,7.121,148.487
C01371=1190.664,259.124,-64.846,-177.108,7.119,148.488
C01372=1190.669,258.876,-64.819,-177.111,7.116,148.488
C01373=1190.673,258.627,-64.791,-177.113,7.114,148.488
C01374=1190.677,258.378,-64.764,-177.116,7.111,148.488
C01375=1190.682,258.130,-64.737,-177.118,7.109,148.488
C01376=1190.686,257.882,-64.710,-177.121,7.106,148.488
C01377=1190.690,257.633,-64.683,-177.123,7.104,148.488
C01378=1190.694,257.385,-64.656,-177.126,7.101,148.488
C01379=1190.699,257.137,-64.628,-177.129,7.099,148.489
C01380=1190.703,256.888,-64.601,-177.132,7.097,148.489
C01381=1190.708,256.640,-64.574,-177.134,7.094,148.489
C01382=1190.713,256.391,-64.547,-177.137,7.092,148.489
C01383=1190.717,256.142,-64.519,-177.139,7.090,148.489
C01384=1190.721,255.894,-64.491,-177.142,7.087,148.489
C01385=1190.726,255.646,-64.464,-177.144,7.085,148.490
C01386=1190.730,255.397,-64.438,-177.147,7.082,148.490
C01387=1190.734,255.149,-64.411,-177.149,7.080,148.490
C01388=1190.739,254.900,-64.384,-177.152,7.077,148.490
C01389=1190.743,254.651,-64.356,-177.155,7.075,148.490
C01390=1190.748,254.403,-64.329,-177.157,7.073,148.490
C01391=1190.752,254.154,-64.302,-177.160,7.070,148.490
C01392=1190.756,253.906,-64.276,-177.162,7.068,148.491
C01393=1190.761,253.658,-64.249,-177.165,7.065,148.491
C01394=1190.765,253.409,-64.222,-177.168,7.063,148.491
C01395=1190.770,253.161,-64.195,-177.170,7.060,148.491
C01396=1190.774,252.911,-64.167,-177.173,7.058,148.491
C01397=1190.778,252.663,-64.141,-177.176,7.055,148.491
C01398=1190.783,252.415,-64.114,-177.178,7.053,148.491
C01399=1190.787,252.166,-64.087,-177.181,7.050,148.492
C01400=1190.792,251.918,-64.059,-177.183,7.048,148.492
C01401=1190.796,251.670,-64.033,-177.186,7.045,148.492
C01402=1190.801,251.421,-64.006,-177.188,7.043,148.492
C01403=1190.805,251.173,-63.979,-177.191,7.041,148.492
C01404=1190.810,250.924,-63.952,-177.194,7.038,148.493
C01405=1190.814,250.676,-63.925,-177.196,7.036,148.493
C01406=1190.819,250.427,-63.898,-177.199,7.033,148.493
C01407=1190.823,250.178,-63.871,-177.201,7.031,148.493
C01408=1190.826,249.930,-63.844,-177.204,7.028,148.493
C01409=1190.831,249.681,-63.817,-177.207,7.027,148.493
C01410=1190.836,249.432,-63.791,-177.209,7.024,148.494
C01411=1190.840,249.184,-63.765,-177.212,7.021,148.494
C01412=1190.845,248.936,-63.737,-177.214,7.020,148.494
C01413=1190.849,248.687,-63.710,-177.217,7.017,148.494
C01414=1190.853,248.439,-63.684,-177.220,7.015,148.494
C01415=1190.858,248.190,-63.658,-177.222,7.012,148.494
C01416=1190.863,247.941,-63.631,-177.225,7.010,148.494
C01417=1190.867,247.693,-63.604,-177.227,7.008,148.495
C01418=1190.871,247.445,-63.577,-177.230,7.005,148.495
C01419=1190.876,247.196,-63.551,-177.233,7.003,148.495
C01420=1190.880,246.947,-63.524,-177.235,7.000,148.495
C01421=1190.885,246.699,-63.497,-177.238,6.998,148.495
C01422=1190.889,246.451,-63.471,-177.241,6.995,148.496
C01423=1190.894,246.202,-63.444,-177.243,6.993,148.496
C01424=1190.898,245.953,-63.418,-177.245,6.991,148.496
C01425=1190.902,245.705,-63.391,-177.248,6.988,148.496
C01426=1190.907,245.456,-63.365,-177.251,6.986,148.496
C01427=1190.911,245.208,-63.338,-177.253,6.983,148.496
C01428=1190.916,244.959,-63.312,-177.256,6.982,148.497
C01429=1190.920,244.710,-63.285,-177.258,6.979,148.497
C01430=1190.924,244.462,-63.259,-177.261,6.977,148.497
C01431=1190.929,244.213,-63.232,-177.264,6.975,148.497
C01432=1190.933,243.965,-63.206,-177.267,6.972,148.497
C01433=1190.939,243.716,-63.180,-177.269,6.970,148.498
C01434=1190.942,243.468,-63.153,-177.271,6.968,148.498
C01435=1190.947,243.219,-63.127,-177.274,6.965,148.498
C01436=1190.951,242.971,-63.101,-177.277,6.963,148.498
C01437=1190.956,242.722,-63.074,-177.280,6.960,148.498
C01438=1190.960,242.474,-63.048,-177.282,6.958,148.498
C01439=1190.965,242.225,-63.021,-177.285,6.956,148.499
C01440=1190.969,241.976,-62.995,-177.287,6.953,148.499
C01441=1190.974,241.727,-62.969,-177.290,6.951,148.499
C01442=1190.978,241.479,-62.942,-177.292,6.949,148.499
C01443=1190.982,241.230,-62.916,-177.295,6.947,148.499
C01444=1190.987,240.982,-62.890,-177.297,6.944,148.500
C01445=1190.992,240.734,-62.864,-177.301,6.942,148.500
C01446=1190.996,240.485,-62.837,-177.303,6.940,148.500
C01447=1191.001,240.236,-62.811,-177.305,6.938,148.500
C01448=1191.005,239.988,-62.785,-177.308,6.935,148.500
C01449=1191.009,239.739,-62.758,-177.311,6.933,148.501
C01450=1191.014,239.490,-62.733,-177.313,6.931,148.501
C01451=1191.018,239.243,-62.707,-177.316,6.928,148.501
C01452=1191.023,238.994,-62.680,-177.318,6.926,148.501
C01453=1191.027,238.745,-62.654,-177.321,6.924,148.501
C01454=1191.031,238.497,-62.628,-177.324,6.921,148.502
C01455=1191.036,238.248,-62.602,-177.326,6.919,148.502
C01456=1191.041,237.999,-62.576,-177.329,6.916,148.502
C01457=1191.045,237.751,-62.550,-177.332,6.915,148.502
C01458=1191.050,237.502,-62.523,-177.334,6.912,148.502
C01459=1191.054,237.253,-62.498,-177.337,6.910,148.503
C01460=1191.059,236.981,-62.470,-177.340,6.908,148.503
C01461=1191.063,236.710,-62.441,-177.342,6.905,148.503
C01462=1191.069,236.439,-62.413,-177.346,6.902,148.503
C01463=1191.074,236.167,-62.384,-177.348,6.900,148.504
C01464=1191.078,235.919,-62.358,-177.351,6.897,148.504
C01465=1191.082,235.670,-62.332,-177.354,6.896,148.504
C01466=1191.087,235.422,-62.307,-177.356,6.893,148.504
C01467=1191.092,235.173,-62.281,-177.359,6.891,148.504
C01468=1191.096,234.924,-62.255,-177.361,6.889,148.505
C01469=1191.100,234.676,-62.228,-177.364,6.887,148.505
C01470=1191.105,234.427,-62.203,-177.367,6.884,148.505
C01471=1191.109,234.179,-62.177,-177.369,6.882,148.505
C01472=1191.114,233.930,-62.151,-177.372,6.880,148.506
C01473=1191.118,233.681,-62.125,-177.375,6.877,148.506
C01474=1191.123,233.433,-62.100,-177.377,6.875,148.506
C01475=1191.127,233.184,-62.074,-177.379,6.873,148.506
C01476=1191.132,232.935,-62.048,-177.382,6.871,148.506
C01477=1191.136,232.686,-62.023,-177.385,6.868,148.506
C01478=1191.141,232.438,-61.997,-177.387,6.867,148.507
C01479=1191.146,232.189,-61.971,-177.390,6.865,148.507
C01480=1191.150,231.940,-61.945,-177.393,6.862,148.507
C01481=1191.155,231.692,-61.920,-177.395,6.860,148.507
C01482=1191.159,231.443,-61.894,-177.398,6.858,148.508
C01483=1191.163,231.194,-61.868,-177.401,6.855,148.508
C01484=1191.168,230.946,-61.843,-177.403,6.853,148.508
C01485=1191.172,230.698,-61.817,-177.406,6.851,148.508
C01486=1191.176,230.449,-61.791,-177.409,6.849,148.509
C01487=1191.181,230.200,-61.766,-177.411,6.846,148.509
C01488=1191.185,229.952,-61.740,-177.414,6.845,148.509
C01489=1191.190,229.703,-61.714,-177.416,6.842,148.509
C01490=1191.194,229.454,-61.689,-177.419,6.840,148.509
C01491=1191.199,229.206,-61.663,-177.422,6.838,148.510
C01492=1191.204,228.956,-61.638,-177.424,6.836,148.510
C01493=1191.209,228.708,-61.612,-177.427,6.833,148.510
C01494=1191.213,228.459,-61.587,-177.429,6.831,148.510
C01495=1191.217,228.211,-61.561,-177.432,6.829,148.511
C01496=1191.222,227.963,-61.535,-177.435,6.826,148.511
C01497=1191.226,227.714,-61.510,-177.437,6.824,148.511
C01498=1191.230,227.465,-61.485,-177.440,6.823,148.511
C01499=1191.235,227.217,-61.460,-177.443,6.821,148.512
C01500=1191.239,226.968,-61.434,-177.445,6.818,148.512
C01501=1191.244,226.720,-61.409,-177.448,6.816,148.512
C01502=1191.249,226.470,-61.384,-177.450,6.814,148.512
C01503=1191.253,226.221,-61.358,-177.453,6.811,148.512
C01504=1191.258,225.973,-61.332,-177.456,6.809,148.513
C01505=1191.262,225.725,-61.307,-177.458,6.807,148.513
C01506=1191.267,225.476,-61.282,-177.461,6.805,148.513
C01507=1191.271,225.227,-61.256,-177.464,6.803,148.514
C01508=1191.275,224.978,-61.231,-177.466,6.801,148.514
C01509=1191.281,224.729,-61.206,-177.469,6.799,148.514
C01510=1191.285,224.481,-61.180,-177.471,6.797,148.514
C01511=1191.289,224.233,-61.155,-177.474,6.794,148.514
C01512=1191.293,223.983,-61.130,-177.477,6.792,148.515
C01513=1191.298,223.735,-61.105,-177.479,6.790,148.515
C01514=1191.303,223.486,-61.080,-177.482,6.788,148.515
C01515=1191.308,223.238,-61.055,-177.485,6.785,148.515
C01516=1191.312,222.989,-61.029,-177.488,6.784,148.516
C01517=1191.316,222.740,-61.004,-177.490,6.781,148.516
C01518=1191.320,222.492,-60.979,-177.492,6.780,148.516
C01519=1191.325,222.242,-60.954,-177.496,6.777,148.516
C01520=1191.330,221.994,-60.929,-177.498,6.775,148.517
C01521=1191.334,221.745,-60.903,-177.500,6.773,148.517
C01522=1191.339,221.497,-60.878,-177.503,6.771,148.517
C01523=1191.343,221.248,-60.854,-177.506,6.768,148.517
C01524=1191.348,221.000,-60.828,-177.508,6.766,148.518
C01525=1191.352,220.750,-60.803,-177.511,6.765,148.518
C01526=1191.357,220.502,-60.778,-177.513,6.762,148.518
C01527=1191.361,220.253,-60.753,-177.516,6.760,148.518
C01528=1191.366,220.005,-60.728,-177.519,6.758,148.519
C01529=1191.370,219.755,-60.703,-177.521,6.756,148.519
C01530=1191.375,219.507,-60.678,-177.524,6.754,148.519
C01531=1191.379,219.258,-60.653,-177.527,6.751,148.519
C01532=1191.384,219.009,-60.628,-177.529,6.749,148.520
C01533=1191.389,218.761,-60.603,-177.532,6.747,148.520
C01534=1191.393,218.512,-60.579,-177.535,6.746,148.520
C01535=1191.398,218.263,-60.554,-177.538,6.743,148.521
C01536=1191.402,218.015,-60.528,-177.540,6.741,148.521
C01537=1191.406,217.766,-60.504,-177.543,6.739,148.521
C01538=1191.411,217.517,-60.479,-177.545,6.737,148.521
C01539=1191.416,217.269,-60.454,-177.548,6.734,148.521
C01540=1191.419,217.020,-60.429,-177.551,6.732,148.522
C01541=1191.425,216.771,-60.405,-177.553,6.731,148.522
C01542=1191.429,216.523,-60.379,-177.556,6.729,148.522
C01543=1191.433,216.274,-60.355,-177.558,6.727,148.523
C01544=1191.438,216.025,-60.330,-177.561,6.724,148.523
C01545=1191.442,215.776,-60.306,-177.564,6.722,148.523
C01546=1191.447,215.528,-60.280,-177.566,6.720,148.523
C01547=1191.452,215.279,-60.256,-177.569,6.718,148.524
C01548=1191.456,215.030,-60.231,-177.572,6.716,148.524
C01549=1191.461,214.781,-60.207,-177.575,6.714,148.524
C01550=1191.465,214.533,-60.182,-177.577,6.712,148.524
C01551=1191.470,214.284,-60.157,-177.580,6.710,148.525
C01552=1191.475,214.035,-60.132,-177.582,6.708,148.525
C01553=1191.479,213.786,-60.108,-177.585,6.705,148.525
C01554=1191.484,213.537,-60.083,-177.588,6.703,148.525
C01555=1191.488,213.289,-60.059,-177.590,6.701,148.526
C01556=1191.493,213.040,-60.034,-177.593,6.700,148.526
C01557=1191.497,212.791,-60.010,-177.596,6.698,148.527
C01558=1191.502,212.542,-59.985,-177.598,6.695,148.527
C01559=1191.506,212.294,-59.960,-177.601,6.693,148.527
C01560=1191.511,212.045,-59.935,-177.604,6.691,148.527
C01561=1191.515,211.797,-59.911,-177.606,6.689,148.528
C01562=1191.520,211.547,-59.886,-177.608,6.687,148.528
C01563=1191.524,211.299,-59.862,-177.612,6.685,148.528
C01564=1191.529,211.029,-59.835,-177.614,6.683,148.528
C01565=1191.535,210.758,-59.809,-177.617,6.681,148.529
C01566=1191.539,210.487,-59.782,-177.620,6.678,148.529
C01567=1191.544,210.217,-59.756,-177.623,6.676,148.529
C01568=1191.549,209.969,-59.732,-177.626,6.674,148.530
C01569=1191.553,209.720,-59.707,-177.628,6.672,148.530
C01570=1191.558,209.471,-59.682,-177.631,6.670,148.530
C01571=1191.562,209.222,-59.658,-177.634,6.668,148.530
C01572=1191.567,208.974,-59.634,-177.636,6.666,148.531
C01573=1191.571,208.724,-59.609,-177.639,6.664,148.531
C01574=1191.576,208.476,-59.585,-177.642,6.661,148.531
C01575=1191.581,208.227,-59.561,-177.644,6.660,148.532
C01576=1191.585,207.978,-59.537,-177.647,6.658,148.532
C01577=1191.590,207.729,-59.512,-177.650,6.656,148.532
C01578=1191.594,207.480,-59.488,-177.652,6.654,148.532
C01579=1191.599,207.232,-59.464,-177.654,6.652,148.533
C01580=1191.604,206.983,-59.439,-177.658,6.649,148.533
C01581=1191.608,206.735,-59.415,-177.660,6.648,148.533
C01582=1191.612,206.485,-59.391,-177.663,6.646,148.534
C01583=1191.617,206.236,-59.367,-177.665,6.644,148.534
C01584=1191.622,205.988,-59.343,-177.668,6.642,148.534
C01585=1191.626,205.740,-59.319,-177.670,6.640,148.534
C01586=1191.632,205.490,-59.295,-177.673,6.638,148.535
C01587=1191.635,205.241,-59.270,-177.676,6.636,148.535
C01588=1191.640,204.993,-59.246,-177.678,6.633,148.535
C01589=1191.644,204.744,-59.222,-177.681,6.632,148.536
C01590=1191.650,204.495,-59.198,-177.684,6.630,148.536
C01591=1191.654,204.247,-59.174,-177.686,6.628,148.536
C01592=1191.658,203.997,-59.150,-177.689,6.626,148.537
C01593=1191.662,203.749,-59.126,-177.692,6.624,148.537
C01594=1191.668,203.500,-59.102,-177.694,6.621,148.537
C01595=1191.672,203.251,-59.078,-177.697,6.620,148.537
C01596=1191.676,203.003,-59.053,-177.700,6.618,148.538
C01597=1191.681,202.754,-59.030,-177.702,6.616,148.538
C01598=1191.685,202.505,-59.006,-177.705,6.614,148.538
C01599=1191.690,202.255,-58.982,-177.707,6.612,148.539
C01600=1191.695,202.007,-58.958,-177.710,6.610,148.539
C01601=1191.699,201.759,-58.934,-177.713,6.608,148.539
C01602=1191.704,201.510,-58.910,-177.716,6.606,148.540
C01603=1191.708,201.261,-58.886,-177.718,6.604,148.540
C01604=1191.714,201.012,-58.862,-177.721,6.602,148.540
C01605=1191.718,200.763,-58.838,-177.723,6.600,148.540
C01606=1191.722,200.514,-58.814,-177.726,6.598,148.541
C01607=1191.727,200.265,-58.790,-177.729,6.596,148.541
C01608=1191.731,200.016,-58.767,-177.731,6.595,148.541
C01609=1191.736,199.768,-58.743,-177.734,6.593,148.542
C01610=1191.740,199.519,-58.719,-177.737,6.590,148.542
C01611=1191.745,199.270,-58.695,-177.740,6.588,148.542
C01612=1191.750,199.021,-58.671,-177.742,6.586,148.543
C01613=1191.755,198.773,-58.647,-177.745,6.584,148.543
C01614=1191.759,198.524,-58.624,-177.747,6.583,148.543
C01615=1191.764,198.275,-58.600,-177.750,6.581,148.544
C01616=1191.768,198.026,-58.577,-177.753,6.579,148.544
C01617=1191.773,197.778,-58.553,-177.755,6.577,148.544
C01618=1191.777,197.529,-58.529,-177.757,6.575,148.544
C01619=1191.782,197.280,-58.506,-177.760,6.573,148.545
C01620=1191.786,197.030,-58.481,-177.763,6.571,148.545
C01621=1191.791,196.781,-58.458,-177.766,6.569,148.545
C01622=1191.795,196.533,-58.434,-177.769,6.567,148.546
C01623=1191.800,196.284,-58.411,-177.771,6.565,148.546
C01624=1191.804,196.035,-58.387,-177.774,6.563,148.546
C01625=1191.809,195.787,-58.363,-177.777,6.562,148.547
C01626=1191.814,195.538,-58.340,-177.779,6.559,148.547
C01627=1191.818,195.288,-58.316,-177.781,6.558,148.547
C01628=1191.823,195.039,-58.293,-177.784,6.556,148.548
C01629=1191.827,194.791,-58.269,-177.787,6.554,148.548
C01630=1191.832,194.542,-58.246,-177.789,6.552,148.548
C01631=1191.837,194.293,-58.222,-177.792,6.550,148.549
C01632=1191.841,194.044,-58.199,-177.795,6.549,148.549
C01633=1191.846,193.796,-58.175,-177.798,6.546,148.549
C01634=1191.851,193.547,-58.151,-177.801,6.544,148.550
C01635=1191.855,193.297,-58.128,-177.803,6.542,148.550
C01636=1191.860,193.048,-58.105,-177.806,6.540,148.550
C01637=1191.865,192.801,-58.081,-177.808,6.538,148.551
C01638=1191.869,192.552,-58.058,-177.811,6.537,148.551
C01639=1191.874,192.303,-58.035,-177.814,6.535,148.551
C01640=1191.878,192.054,-58.012,-177.816,6.533,148.552
C01641=1191.883,191.805,-57.988,-177.819,6.531,148.552
C01642=1191.888,191.556,-57.965,-177.821,6.529,148.552
C01643=1191.892,191.307,-57.941,-177.824,6.528,148.553
C01644=1191.897,191.058,-57.917,-177.826,6.526,148.553
C01645=1191.901,190.809,-57.894,-177.829,6.524,148.553
C01646=1191.905,190.561,-57.871,-177.832,6.522,148.553
C01647=1191.910,190.312,-57.848,-177.834,6.520,148.554
C01648=1191.915,190.063,-57.825,-177.837,6.518,148.554
C01649=1191.920,189.814,-57.801,-177.840,6.517,148.555
C01650=1191.925,189.565,-57.778,-177.842,6.515,148.555
C01651=1191.930,189.316,-57.755,-177.846,6.512,148.555
C01652=1191.934,189.068,-57.732,-177.848,6.510,148.556
C01653=1191.938,188.818,-57.709,-177.851,6.509,148.556
C01654=1191.943,188.569,-57.685,-177.854,6.507,148.556
C01655=1191.948,188.320,-57.662,-177.856,6.505,148.557
C01656=1191.952,188.072,-57.639,-177.858,6.503,148.557
C01657=1191.956,187.823,-57.616,-177.861,6.501,148.557
C01658=1191.962,187.574,-57.593,-177.864,6.499,148.557
C01659=1191.966,187.325,-57.570,-177.866,6.497,148.558
C01660=1191.970,187.077,-57.547,-177.869,6.496,148.558
C01661=1191.975,186.828,-57.523,-177.872,6.494,148.559
C01662=1191.980,186.579,-57.500,-177.874,6.492,148.559
C01663=1191.985,186.329,-57.477,-177.877,6.490,148.559
C01664=1191.989,186.080,-57.455,-177.880,6.488,148.560
C01665=1191.994,185.832,-57.432,-177.882,6.487,148.560
C01666=1191.999,185.583,-57.408,-177.885,6.485,148.560
C01667=1192.003,185.334,-57.386,-177.888,6.483,148.561
C01668=1192.008,185.064,-57.361,-177.890,6.481,148.561
C01669=1192.013,184.795,-57.335,-177.893,6.479,148.561
C01670=1192.018,184.525,-57.311,-177.896,6.477,148.562
C01671=1192.023,184.255,-57.286,-177.899,6.475,148.562
C01672=1192.027,184.007,-57.263,-177.902,6.473,148.562
C01673=1192.032,183.758,-57.240,-177.904,6.471,148.563
C01674=1192.037,183.509,-57.217,-177.907,6.470,148.563
C01675=1192.041,183.260,-57.195,-177.910,6.468,148.563
C01676=1192.046,183.011,-57.171,-177.912,6.466,148.564
C01677=1192.051,182.762,-57.148,-177.915,6.464,148.564
C01678=1192.055,182.513,-57.125,-177.918,6.462,148.565
C01679=1192.060,182.264,-57.103,-177.920,6.461,148.565
C01680=1192.064,182.015,-57.080,-177.923,6.459,148.565
C01681=1192.069,181.766,-57.057,-177.926,6.457,148.566
C01682=1192.073,181.518,-57.034,-177.928,6.455,148.566
C01683=1192.079,181.269,-57.012,-177.931,6.453,148.566
C01684=1192.083,181.020,-56.989,-177.934,6.452,148.567
C01685=1192.087,180.770,-56.967,-177.936,6.450,148.567
C01686=1192.092,180.521,-56.943,-177.939,6.448,148.567
C01687=1192.097,180.273,-56.921,-177.942,6.446,148.568
C01688=1192.102,180.024,-56.898,-177.944,6.444,148.568
C01689=1192.106,179.775,-56.875,-177.947,6.443,148.568
C01690=1192.111,179.527,-56.852,-177.950,6.441,148.569
C01691=1192.115,179.277,-56.830,-177.952,6.439,148.569
C01692=1192.120,179.028,-56.807,-177.955,6.437,148.570
C01693=1192.124,178.779,-56.785,-177.958,6.435,148.570
C01694=1192.130,178.531,-56.762,-177.960,6.434,148.570
C01695=1192.134,178.281,-56.740,-177.962,6.433,148.571
C01696=1192.139,178.032,-56.716,-177.965,6.431,148.571
C01697=1192.143,177.784,-56.695,-177.968,6.429,148.571
C01698=1192.148,177.534,-56.671,-177.970,6.427,148.572
C01699=1192.152,177.286,-56.649,-177.973,6.426,148.572
C01700=1192.157,177.037,-56.627,-177.976,6.424,148.572
C01701=1192.162,176.787,-56.604,-177.978,6.422,148.573
C01702=1192.166,176.539,-56.582,-177.981,6.420,148.573
C01703=1192.172,176.290,-56.559,-177.984,6.418,148.574
C01704=1192.175,176.041,-56.537,-177.986,6.417,148.574
C01705=1192.180,175.791,-56.514,-177.989,6.415,148.574
C01706=1192.185,175.543,-56.492,-177.992,6.413,148.575
C01707=1192.189,175.294,-56.469,-177.994,6.411,148.575
C01708=1192.195,175.046,-56.446,-177.997,6.409,148.575
C01709=1192.199,174.796,-56.424,-178.000,6.408,148.576
C01710=1192.203,174.547,-56.402,-178.002,6.406,148.576
C01711=1192.208,174.299,-56.379,-178.005,6.404,148.576
C01712=1192.213,174.049,-56.357,-178.008,6.402,148.577
C01713=1192.217,173.800,-56.335,-178.010,6.400,148.577
C01714=1192.222,173.552,-56.312,-178.013,6.400,148.578
C01715=1192.227,173.302,-56.290,-178.015,6.398,148.578
C01716=1192.231,173.054,-56.269,-178.018,6.396,148.578
C01717=1192.236,172.805,-56.245,-178.021,6.394,148.579
C01718=1192.241,172.556,-56.224,-178.023,6.392,148.579
C01719=1192.245,172.307,-56.201,-178.026,6.391,148.579
C01720=1192.250,172.057,-56.179,-178.029,6.389,148.580
C01721=1192.255,171.809,-56.156,-178.031,6.387,148.580
C01722=1192.259,171.560,-56.134,-178.034,6.385,148.580
C01723=1192.265,171.311,-56.112,-178.037,6.383,148.581
C01724=1192.269,171.061,-56.090,-178.039,6.382,148.581
C01725=1192.274,170.813,-56.068,-178.042,6.380,148.582
C01726=1192.278,170.564,-56.046,-178.044,6.379,148.582
C01727=1192.283,170.315,-56.023,-178.047,6.377,148.582
C01728=1192.288,170.066,-56.001,-178.049,6.375,148.583
C01729=1192.292,169.816,-55.979,-178.053,6.374,148.583
C01730=1192.296,169.568,-55.957,-178.055,6.372,148.584
C01731=1192.301,169.319,-55.935,-178.058,6.370,148.584
C01732=1192.306,169.070,-55.913,-178.061,6.368,148.584
C01733=1192.311,168.821,-55.890,-178.063,6.367,148.585
C01734=1192.316,168.572,-55.869,-178.066,6.365,148.585
C01735=1192.320,168.323,-55.847,-178.069,6.363,148.585
C01736=1192.325,168.074,-55.825,-178.071,6.361,148.586
C01737=1192.330,167.824,-55.802,-178.073,6.360,148.586
C01738=1192.335,167.576,-55.781,-178.076,6.359,148.587
C01739=1192.338,167.327,-55.758,-178.079,6.357,148.587
C01740=1192.343,167.078,-55.736,-178.081,6.355,148.587
C01741=1192.348,166.830,-55.715,-178.084,6.353,148.588
C01742=1192.352,166.581,-55.693,-178.087,6.351,148.588
C01743=1192.357,166.332,-55.671,-178.089,6.350,148.588
C01744=1192.362,166.082,-55.648,-178.093,6.348,148.589
C01745=1192.367,165.834,-55.627,-178.095,6.347,148.589
C01746=1192.372,165.584,-55.604,-178.097,6.345,148.590
C01747=1192.376,165.336,-55.583,-178.100,6.344,148.590
C01748=1192.381,165.086,-55.561,-178.103,6.342,148.590
C01749=1192.386,164.838,-55.539,-178.105,6.340,148.591
C01750=1192.390,164.588,-55.517,-178.108,6.338,148.591
C01751=1192.395,164.339,-55.496,-178.111,6.337,148.592
C01752=1192.400,164.090,-55.474,-178.113,6.335,148.592
C01753=1192.404,163.841,-55.452,-178.116,6.334,148.592
C01754=1192.409,163.592,-55.431,-178.118,6.332,148.593
C01755=1192.413,163.343,-55.409,-178.121,6.331,148.593
C01756=1192.418,163.094,-55.387,-178.124,6.329,148.594
C01757=1192.422,162.845,-55.365,-178.127,6.327,148.594
C01758=1192.427,162.596,-55.343,-178.129,6.325,148.594
C01759=1192.432,162.348,-55.322,-178.132,6.323,148.595
C01760=1192.437,162.098,-55.300,-178.134,6.322,148.595
C01761=1192.442,161.849,-55.278,-178.137,6.321,148.596
C01762=1192.446,161.601,-55.257,-178.140,6.319,148.596
C01763=1192.451,161.351,-55.235,-178.142,6.317,148.596
C01764=1192.456,161.103,-55.213,-178.145,6.315,148.597
C01765=1192.460,160.853,-55.192,-178.148,6.314,148.597
C01766=1192.465,160.604,-55.170,-178.151,6.312,148.598
C01767=1192.470,160.355,-55.148,-178.153,6.311,148.598
C01768=1192.474,160.106,-55.126,-178.155,6.309,148.598
C01769=1192.479,159.857,-55.105,-178.158,6.308,148.599
C01770=1192.484,159.608,-55.084,-178.161,6.306,148.599
C01771=1192.488,159.359,-55.062,-178.164,6.304,148.599
C01772=1192.493,159.090,-55.039,-178.167,6.303,148.600
C01773=1192.498,158.821,-55.015,-178.169,6.301,148.600
C01774=1192.503,158.552,-54.992,-178.172,6.299,148.601
C01775=1192.509,158.283,-54.969,-178.175,6.297,148.601
C01776=1192.513,158.034,-54.947,-178.178,6.296,148.602
C01777=1192.519,157.785,-54.926,-178.181,6.294,148.602
C01778=1192.524,157.536,-54.904,-178.183,6.293,148.603
C01779=1192.527,157.287,-54.883,-178.185,6.291,148.603
C01780=1192.532,157.038,-54.862,-178.188,6.290,148.603
C01781=1192.537,156.789,-54.840,-178.191,6.288,148.604
C01782=1192.541,156.540,-54.818,-178.193,6.286,148.604
C01783=1192.547,156.290,-54.797,-178.197,6.285,148.605
C01784=1192.551,156.042,-54.776,-178.199,6.284,148.605
C01785=1192.556,155.793,-54.755,-178.201,6.282,148.605
C01786=1192.560,155.544,-54.733,-178.204,6.280,148.606
C01787=1192.565,155.294,-54.712,-178.207,6.278,148.606
C01788=1192.570,155.046,-54.690,-178.209,6.276,148.607
C01789=1192.575,154.796,-54.670,-178.211,6.275,148.607
C01790=1192.579,154.547,-54.648,-178.215,6.274,148.608
C01791=1192.584,154.299,-54.626,-178.217,6.272,148.608
C01792=1192.589,154.049,-54.605,-178.220,6.271,148.608
C01793=1192.594,153.800,-54.584,-178.223,6.269,148.609
C01794=1192.598,153.551,-54.562,-178.225,6.268,148.609
C01795=1192.603,153.302,-54.542,-178.227,6.266,148.609
C01796=1192.608,153.053,-54.520,-178.231,6.265,148.610
C01797=1192.613,152.804,-54.499,-178.233,6.263,148.610
C01798=1192.616,152.555,-54.478,-178.236,6.261,148.611
C01799=1192.622,152.306,-54.457,-178.238,6.260,148.611
C01800=1192.626,152.057,-54.435,-178.241,6.258,148.612
C01801=1192.632,151.808,-54.414,-178.243,6.256,148.612
C01802=1192.636,151.559,-54.394,-178.247,6.255,148.613
C01803=1192.640,151.310,-54.372,-178.249,6.254,148.613
C01804=1192.645,151.060,-54.351,-178.251,6.252,148.613
C01805=1192.650,150.811,-54.331,-178.254,6.251,148.614
C01806=1192.655,150.563,-54.309,-178.257,6.249,148.614
C01807=1192.660,150.313,-54.288,-178.259,6.247,148.614
C01808=1192.664,150.065,-54.267,-178.262,6.246,148.615
C01809=1192.669,149.815,-54.245,-178.265,6.245,148.615
